# B&R Automation Studio project NAEUL004C00R13L518F00 (part 6)

### Hardware
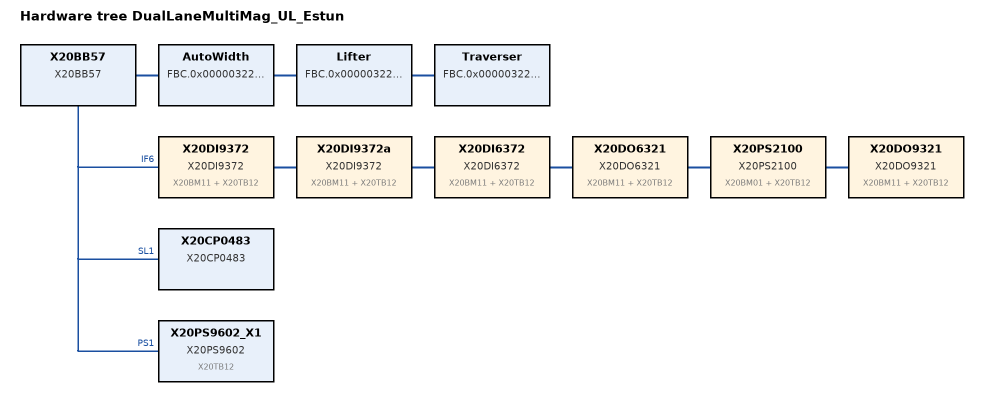
[picture p16: hardware tree DualLaneMultiMag_UL_Estun]
```
AutoWidth : FBC.0x00000322.0x00001000.NUTEK_ESTUN_PronetPlus_EDS_V106 v1.06.1 (OrderNumber=NUTEK_ESTUN_PronetPlus_V106)  [CAN1 -> X20BB57.IF7 (NodeNumber=16)]
Lifter : FBC.0x00000322.0x00001000.NUTEK_ESTUN_PronetPlus_EDS_V106 v1.06.1 (OrderNumber=NUTEK_ESTUN_PronetPlus_V106)  [CAN1 -> AutoWidth.CAN2 (NodeNumber=17)]
Traverser : FBC.0x00000322.0x00001000.NUTEK_ESTUN_PronetPlus_EDS_V106 v1.06.1 (OrderNumber=NUTEK_ESTUN_PronetPlus_V106)  [CAN1 -> Lifter.CAN2]
X20BB57 : X20BB57 v1.1.1.0
  Connector IF1:
    Baudrate = 9600
    Parity = N
  Connector IF7:
    Baudrate = 1000000
    ActivateCanOpen = 1
    p100c_parametervalue = 1000
    p100d_parametervalue = 3
X20BM01 : X20BM01 v2.1.0.0  [X2X1 -> X20BM11e.X2X2]
X20BM11 : X20BM11 v1.0.0.1  [X2X1 -> X20BB57.IF6]
X20BM11a : X20BM11 v1.0.0.1  [X2X1 -> X20BM11.X2X2]
X20BM11b : X20BM11 v1.0.0.1  [X2X1 -> X20BM11a.X2X2]
X20BM11e : X20BM11 v1.0.0.1  [X2X1 -> X20BM11b.X2X2]
X20BM11f : X20BM11 v1.0.0.1  [X2X1 -> X20BM01.X2X2]
X20CP0483 : X20CP0483 v1.2.1.0  [SL -> X20BB57.SL1]
  Connector IF2:
    ActivateDevice = 1
    Mode = Manual
    InternetAddress = 192.168.0.14
    SubnetMask = 255.255.255.0
    InaNodeNumber = 14
    Vnc1
    VncVcObjectName1 = Visu
    VncKeyMappingFile1 = 
    VncMaxConnections1 = 3
    VncRefreshRate1 = 100
    ActivateSnmp = 2
  ConfigurationID = NAEUL004
  VolatileGlobalPvSize = 80000
  EnableUsbRemoteInstall = 1
  TimerDeviceType = SWIOTIMER
  Cyclic1Duration = 10000
  Cyclic1Tolerance = 10000
  Cyclic2Duration = 20000
  Cyclic2Tolerance = 20000
  Cyclic3Duration = 50000
  Cyclic3Tolerance = 50000
  Cyclic4Duration = 10000
  Cyclic4Tolerance = 10000
  Cyclic5Duration = 200000
  Cyclic5Tolerance = 200000
  Cyclic6Duration = 500000
  Cyclic6Tolerance = 500000
  Cyclic7Duration = 1000000
  Cyclic7Tolerance = 1000000
  Cyclic8Duration = 10000
  Cyclic8Tolerance = 10000
  FileDevice1
  FileDeviceName1 = C
  FileDevicePath1 = C:
  FileDevice2
  FileDeviceName2 = User
  FileDevicePath2 = C:\User
  FileDevice3
  FileDeviceName3 = Private
  FileDevicePath3 = C:\Private
  FileDevice4
  FileDeviceName4 = CustomerUser
  FileDevicePath4 = C:\User\UserMgmt
  FileDevice5
  FileDeviceName5 = ProdRcp
  FileDevicePath5 = C:\User\ProductRecipe
  FileDevice6
  FileDeviceName6 = MagRcp
  FileDevicePath6 = C:\User\MagazineRecipe
  FileDevice7
  FileDeviceName7 = Alarm
  FileDevicePath7 = C:\User\Alarm
  FileDevice8
  FileDeviceName8 = McParam
  FileDevicePath8 = C:\User\MachineParameter
  FileDevice9
  FileDeviceName9 = NtParam
  FileDevicePath9 = C:\Private\NutekParameter
  FileDevice10
  FileDeviceName10 = LibVer
  FileDevicePath10 = C:\User\LibrariesVersion
  FileDevice11
  FileDeviceName11 = Retain
  FileDevicePath11 = C:\User\Retain
  FileDevice12
  FileDeviceName12 = Log
  FileDevicePath12 = C:\User\Log
  FileDevice13
  FileDeviceName13 = LCS
  FileDevicePath13 = C:\User\LCS
  FileDevice14
  FileDeviceName14 = MpProdRcp
  FileDevicePath14 = C:\User\ProductRecipeXml
  FileDevice15
  FileDeviceName15 = MpNtParam
  FileDevicePath15 = C:\Private\NutekParameterXml
  FtpUser1
  FtpUsername1 = NTAFTP
  FtpUserPassword1 = +UZ5u8Axw7KkkY4oM/r7wOOfB5oWHxpSY6r3j++jJso=  // NTA4BH
  FtpUserSalt1 = c0Alfi1W
  FTPAccessRight1 = 0
  FTPdevice1 = ALL
  FtpUser2
  FtpUsername2 = admin
  FtpUserPassword2 = mW+qRsE1LOSFDAB60rBJwb9dZ7uQUIuoHZp04C+x5XU=  // admin
  FtpUserSalt2 = Nr9+IHjr
  FTPAccessRight2 = 0
  FTPMSPartition2 = SYSTEM
  FTPMSpath2 = User
  FtpUser3
  FtpUsername3 = LCS
  FtpUserPassword3 = W4lkF6NjcyaB1sRdLwIoSAlqHoAE4GimWQdq7pKTzbA=  // LCS
  FtpUserSalt3 = f3H7b7h0
  FTPMSPartition3 = SYSTEM
  FTPMSpath3 = User\LCS
  ActivateOpcUa = 1
  OpcUa_ConversationSecurityPolicy_EnableBasic256Rsa256 = 0
  OpcUaInformationModels_PV_Version = 1
X20DI6372 : X20DI6372 v1.1.0.0  [SS1 -> X20TB12c.SS; SL -> X20BM11b.SL1]
X20DI9372 : X20DI9372 v1.1.0.0  [SS1 -> X20TB12a.SS; SL -> X20BM11.SL1]
X20DI9372a : X20DI9372 v1.1.0.0  [SS1 -> X20TB12b.SS; SL -> X20BM11a.SL1]
X20DO6321 : X20DO6321 v1.1.0.0  [SS1 -> X20TB12f.SS; SL -> X20BM11e.SL1]
X20DO9321 : X20DO9321 v1.1.0.0  [SS1 -> X20TB12h.SS; SL -> X20BM11f.SL1]
X20PS2100 : X20PS2100 v1.2.0.0  [SS1 -> X20TB12g.SS; SL -> X20BM01.SL1]
X20PS9602_X1 : X20PS9602 v1.0.2.0  [PS -> X20BB57.PS1; SS1 -> X20TB12.SS]
X20TB12 : X20TB12 v1.0.0.0
X20TB12a : X20TB12 v1.0.0.0
X20TB12b : X20TB12 v1.0.0.0
X20TB12c : X20TB12 v1.0.0.0
X20TB12f : X20TB12 v1.0.0.0
X20TB12g : X20TB12 v1.0.0.0
X20TB12h : X20TB12 v1.0.0.0
```

## Logical view

Binary libraries used (declarations not repeated): standard, runtime, astime, asstring, operator, AsIecCon, AsCANopen, visapi, FileIO, AsIODiag, AsMem, dvframe, AsOpcUac, AsARCfg, sys_lib, AsTCP, AsFltGen, brsystem, MpCom, MpBase, MpRecipe, Acp10man, Acp10par, NcGlobal, AsMath, NtBuffer, NtConv, NtFileIO, NtLogFile, NtMem, NtMessage, NtOvenInfo, NtPneu, NtRS232, NtSMEMA, NtTCP, NtTLBuz, NtVersion, NtSOT 5.00.0, NtLF, NtMotion, NtRecipe 5.00.5, NtHermes 5.00.4, NtOPCUA 5.00.1

### Update LogLibrary.txt
```
2023-09-06
NtOPCUA 6.01.0 - Add fbOPCUAMethodGetHandle and fbOPCUAMethodCall, updated fbOPCUAGetNodeHdlList

2023-05-22
NtHermes 5.00.4 Upgrade the Supervisory Hermes

2022-07-05
NtRecipe 5.00.4 Debug of Sorting Function

2022-01-25
NtRecipe 5.00.4 - Improve fRecipeNmCompare

2021-12-29
NtLF 5.01.5 - Add bDBAOnWOAlign to send DBA even width check sensor is not aligned.

2021-10-19
NtMotion 5.00.9 - Uncheck servo on and homing operation if both have been done.

2021-09-30
NtHermes 5.00.4 - Hermes v1.3

2021-09-01
NtLF 5.01.4 - Modify Product Recipe Name Related Variables to STRING[254].
NtUSB 5.00.5 - Add bEn := false for each fb when they are idling.

2021-07-08
NtUSB 5.00.4 - Improve fbDecodeStdKey.Changed ReadIdx Size, Check Array Limit.

2021-06-28
NtUI 5.00.2 - Add tyUIBitmap & tyUIBtn (uiValueIdx) to accomodate higher range of bitmap offset index

2021-04-20
NtLF 5.01.3 - Update fLFUSAllow & fLFDSAllow Block Conditions
			- Modify fLFFollowerProdAccDataReq.

2021-02-26
NtSMEMA:5.00.6 - Add fbSMEMATransporting1 for DS
NtLF:5.01.2 - Two Modes For Sequential. Modify fLFUSAllow For 3rd Party Usage.

2021-02-24
NtLF:5.01.2 - Modify fLFUSAllow.

2021-02-17
NtMotion 5.00.8 - Limit sensor interlock for Estun Servo Movement. (20210217)
       - Homing timeout in 3 sec if home sensor broken.
       - Set default value for servo parameter if the NtParam setting out of the limit.

2021-02-24
NtLF:5.01.2 - Modify fLFUSAllow.

2021-02-21
NtSMEMA: 5.00.6 - Add fbSMEMATransporting1.

2021-02-17
5.00.8 - Limit sensor intelock for Estun Servo Movement. (20210217)
       - Homing timeout in 3 sec if home sensor broken.
       - Set default value for servo parameter if the NtParam setting out of the limit.

2021-02-05
NtSMEMA:5.00.5 - Update fbSMEMATransporting

2020-11-14
NtUSB 5.00.0 - New Library Design.

2020-11-10
NtMotion:5.00.7 - Torque limit setting at NtParam.

2020-10-05
NtLF:5.01.1 - Improve Change All For Section Leader, Debug Change Sequential.

2020-09-10
NtTCP:5.00.2 - Change of fbTCPClntConnect.

2020-08-17
NtVersion:5.01.1 - Change of fChkFileValidity & fInvalidCharInFileChk to function block.

2020-08-06
NtLF:5.01.0 - Improve leader follower concept.
			- Add more tags in tyLeaderToFollowerTag and tyFollowerToLeaderTag.
NtVersion:5.01.0 - Add fChkFileValidity and fInvalidCharInFileChk.

2020-07-24
NtRecipe:5.00.3 - Debug of sorting functions.

2020-06-30
NtMotion:5.00.6 - Homing action when remote side limit sensor is on.

2020-06-15
NtMotion:5.00.5 - Homing timeout error when limit switch disconnecte.

2020-06-08
NtRecipe:5.00.2 - Update Product Recipe to 254, Add Sorting and End Character Filter Functions.
NtVersion:5.00.1 - Debug of fChkLibrariesVer.

2020-06-07
NtUI:5.00.1 - Update fbTableCtrl and fbTableCtrl_v2. Update tyUILString.

2020-06-01
NtStepper:5.00.0  - New Release.
NtConv:5.00.3	  - Added fbConvSenToSenBrkTm2Lmt & fbConvSenToSenBrk2.

2020-03-20
NtMotion - Add Estun Pronet, Schneider Electric Lexium 28 Servo Motor Control.
		- Resolve Limit Switch Alarm when Delta servo motor perform homing at stratup of auto mode.
NtParam - Add the selection of Motor model.

2020-03-16
NtTLBuz - Add inputs to allow repeat sequence for fbTLBuzWarn.
TLBuz - Add two inputs for buzzer behaviour, towerlight flash function to act_background and reset fbwarning.

2019-12-24
NtLF - Modify fbLeaderBlkDS, include machine index before & after oven 2, block machine to machine when different width
LFLeader - Remove fbBlkDS2 in Act_Initial & Act_Background_Process, add pa_bLFOnline in Act_Background_Process

2019-10-31
TLBuz - Regroup Structure Into Nutek, Aptiv & MEK.
MagConv - Separate Program Into MagConv1Clamper & MagConv2Clamper.

2019-10-29
NtHermes - Debug of fHermesGetTimeStamp

2019-10-21
NtRecipe - Debug Of fRecipeGetInfo.
NtSMEMA - fbSMEMAUS_9851, fbSMEMAUS_Std, fbSMEMADS_OppFirst, reset signal while error.
NtBuffer - Debug of fBffrSetFull, fBffrSetMty for slot disable.
NtLF - Add bBypassMnlAccDat Tag Name, Improve Change All Function Without Manually Accept Data.
MagConv - Improve with Action MagConvActPreExit & MagConvActPreExitClpr.
LFFollower - Improve Change All Function Without Manually Accept Data.
LFLeader - Add Second Oven Index, Improve Change All Function Without Manually Accept Data.
OpcUaMap.uad - Enable bBypassMnlAccDat Tag Name.
Startup - Act_Main_SDOWrite, Remove SDOWrite.
CANOpenServo - Change Structure Of SDOWrite And Abnormal Movement.

2019-07-30
NtMotion - Add Input To Select Homing Without Index Pulse.
CANOpenServo - Due To Upgrade of NtMotion.

2019-07-19
NtSMEMA - fbSMEMADS, reset signal while error.

2019-07-18
LFFollower - Act_Link, Minor debug.

2019-07-15
LCS - Act_Link, Check Recipe Name Must Not Exceed 15 Char.

2019-07-10
LCS - Add More Parameter For Live Data.

2019-07-04
LFFollower - Improve of Recipe Compare Method For p_tyInternalReqProdRcp, tyUpdtProdRcp & tyRlsBrdProdRcpNm.

2019-07-03
LFFollower - Improve Act_Background To Check Whole Product Recipe Different Instead of Name & Width Only.
Buffer - Add p_tyBufferStat & p_tyDispBuffer And Improve For Two Program Control One Memory.
NtBuffer - Debug Of Limit Buffer Range.

2019-06-28
USHermes - Improve of Act_Background_AccData.
DSHermes - Move of Act_Background_ChgConfig.
Buffer - Improve of bParamDiff Condition.
LCSLF - Improve of LCSActRunProd.

2019-06-27
LFFollower - Improvement To Change Name & Width To Whole Product Recipe Type.

2019-06-17
Conv - Add Two Action : ConvActEntToInOff & ConvActRevImmedStart.

2019-06-12
LFFollower - Add Act_Background_ChkRlsBrd. Improvement of Act_Background_UpdtData.
LCSLF - Add Update Data in Act_Background.

2019-06-11
TLBuz - Modify ChgRcp.
LFFollower - Improvement of UpdtData.

2019-06-10
ProdRcp - Update tyCurrRcp To a_tyCurrRcp (Array).
LFFollower - Add p_bInternalUse.
USHermes - Add p_bInternalUse.
DSHermes - Add p_bInternalUse.

2019-06-07
NtTLBuz - Improve of fbTLBuzWarn.
TLBuz - Add Warning & ChgRcp.
TCP - Add Start Code & End Code Checking.
Buffer - Improve bParamDiff. Add bFIFOOld.

2019-06-04
USHermes - Improvement At Accept Date (Act_Background_AccData).

2019-06-02
TCP - New.

2019-05-30
Hermes - Debug CheckAlive. SequenceTO Start Only After Connection Establish.
NtSMEMA - Improve fbSMEMATransportIdle.
Flatstream - Debug Act_Main.
USHermes - Update Act_Link to Accept New Recipe.

2019-05-29
NtRS232 - Add Flatstream Function.
DVFrame - Change From RS232. Improvement & Debug.
Flatstream - New.

2019-05-28
MagConv - Add MagConvActInitClpStop.
DCConv - Improvement of DC Motor Alarm Trigger Time.
LFFollower - Improve of Act_Background.
NtBuffer - Debug of fBffrNxtLoadNearby.
LCS - Add "Warning" & "Info" For Live Data.

2019-05-27
LFFollower - Debug Act_Link.
LCS - Debug Act_Link. Add sErrMsg.
Buffer - Debug Act_Main_Bffr. Add bMagRemoved.
Data - Update of Default User.dat.

2019-05-24
LFFollower - Improve of Act_Background.
MagConv - Add MagConvActEntClpStop.
TLBuz - Modify Warning Condition.

2019-05-22
NtLF - ChgAll Will Bypass Width Check Sensor.
OpcUaMap.uad - Update Tag Name.
LF - Modify Set Time. Improve Of Act_Background for Accept Data.
LFLeader - Add New Tag Name.
Time - Update of Act_InitGlobal For LF Sync Time.
LCS - Update To Reset If Receive Idle From LCS.

2019-05-21
NtRS232 - Add fbFullReadUntilValid.
RS232 - Add FullReadUntilValid.
LCS - Move Some Program From Act_Background To Act_Link. Bug Fixed.

2019-05-20
RS232 - Modify to work with start code & end code.
ProdRcp - Modify on dtLastModified in Act_LinkAction.
LCS - Act_Background Show Boolean & dtLastModified Working Sample. Add Function Enable.
TLBuz - Add Aptiv Mode.
NtParam - Add eTLBuzMod.

2019-05-18
Buffer - Check Next Unload Ignore Product Name.

2019-05-17
NtMessage - Debug When Attribute Value Is Empty String.

2019-05-15
OvenInfo - Improve of Act_Background.
Buffer - Add bParamDiff to check current parameter and request parameter different.

2019-05-14
LCS - Update Act_InitGlobal.
RS232 - New.

2019-05-11
LFFollower - Improve And Able To Ignore MagRcp If Necessary.

2019-05-10
TLBuz - Add Simulation Mode.
ProdRcp - Improve Act_LinkAction.
Buffer - Improve Act_LinkAction.
HWInfo - Improve Act_Main While In Simulation.

2019-05-09
CANOpenServo - Improve of Error Axis Move Abnormally By External Force (10000).
ProdRcp - Debug Write Recipe. Add Save List.
MagRcp - Debug Write Recipe. Add Save List.
UsrFolder - Create LCS Directory.
Startup - Act_Main_UsrFolder, Create LCS Directory.
Alarm - Combine Two Alarm Info.

2019-05-08
RmtHermes - Debug Log title.
UsrMgmt - Add Access Right Output.

2019-05-07
NtConv - After Time Out, Reset Output.
MagConv - Debug.
ConvBffr - Add Individual Have Board Output.
NtLF - Debug fLFUSAllow. Modify fbLFFollower.
LF - Major update.
LCSLF - Change Name to tyCurrProdRcp.
ProdRcp - Add Write Recipe Parameter.
MagRcp - Add Write Recipe Parameter.
LCS - Update to match LCS (PC).

2019-05-04
MagRcp - Split Current Magazine Recipe From McParam.
ProdRcp - Split Current Product Recipe From McParam.
UsrMgmt - Split Access Right From McParam. Remove Nutek User.
Hermes - Split Configuration From McParam. Add RmtHermes.
Startup - Split Parameters From McParam. Add RmtHermes.
Remove "File Device" "NutekUser". Please Refer Configuration "4PPC30_043F_21F001".
NtHermes - Debug Due to RmtHermes.

2019-05-01
Hermes - Log file change to day instead of hour. Due to startup too long to check old log when production run for long.

2019-04-30
LCS - Improve To Match LCS (PC).
LFLeader - Make a_tyFollowerToLeaderTag as Output.
All - sStatTxt & a_sStatText Change To String[200].
ProdRcp - Modify For LCS.

2019-04-28
MpProdRcp - New.
Add "Config.mprecipexml" Under Configuration View > mapp. Please Refer Configuration "4PPC30_043F_21F001".
Add "File devices" For "MpProdRcp". Please Refer Configuration "4PPC30_043F_21F001".
Startup - Modify Due To MpProdRcp.

2019-04-27
NtSMEMA - Improve Standard SMEMA According to Nutek Standard.
DSSMEMA - Update due to NtSMEMA upgrade.

2019-04-26
Buffer - Debug tyBuffer to p_tyBuffer. Improve bLastProductUnload Condition In Unload Board.
Startup - Get Retain ConvBffr.
ConvBffr - Update Link with Startup. Improve bLastProduct Condition In Remove Board. Add Have Board Output.
LFFollower - Improve Act_LinkEn. Add Condition in Act_Link to update current recipe into leader tag.

2019-04-25
NtHermes - Debug fHermesIllegalMsgBrdAvlDS. To Handle MachineReady & StartTransport Send In One Message.
LibVer - Modify To Move LibVer From "Private" To "User".
Update "File devices" For "LibVer". Please Refer Configuration "4PPC30_043F_21F001".
Add "File devices" For "LCS". Please Refer Configuration "4PPC30_043F_21F001".
Modify "FTP Server" "Users". Please Refer Configuration "4PPC30_043F_21F001".
Modify "OpcUaMap.uad". Please Refer Configuration "4PPC30_043F_21F001".
LFLeader - Improvement.

2019-04-24
CANOpenServo - Add actual limit sensor output.
ProdRcp - Add "Add" & "Edit" action. Improve of Act_LinkAction to suit LCS.
LCS - New.

2019-04-23
NtLF - Major upgrade.
LFLeader - New.

2019-04-21
USHermes - Modify Alarm Info.
LFFollower - New.

2019-04-18
ConvBffr - New.
NtBffr - Add Buffer Name, Product Name & Barcode.
Buffer - Change of NtBffr.

2019-04-17
CANOpenServo - Remove Extra Homing Parameter, All Use Under tyMotionCANParamInHm.

2019-04-16
Operations - Remove Accept Data & New Data.
Hermes - Debug Log File. Modify Accept Data.

2019-04-11
USHermes - Debug Log by adding step. Add p_bAccDataRdy.
DSHermes - Debug Log by adding step.
NtConv - Debug of Time Out Error.

2019-04-10
Startup - bNtSettingsLoadDone should be FALSE as default.

2019-04-09
Ops2 - Update of p_bAccDat interlock by Ops1.
USHermes - Update AccDatStep in Act_Link. Remove p_bChkBrdAvl. eStatus2 = Error then bRdyRcv = false. Update Act_Background_BoardAvailableChk. Add Manual Accept Data.
DSHermes - Make local.var BoardAvailable new board parameter to default value.
NtParam - Change of Act_LinkAction.
TLBuz - Change of Act_LinkAction.
Buffer - Change of Act_LinkAction.
Conv - Change of Act_LinkAction.
DCConv - Change of Act_LinkAction.
MagConv - Change of Act_LinkAction.
MotorBrk - Change of Act_LinkAction.
ConvSpd - Change of Act_LinkAction.
SMEMA - Change of Act_LinkAction.
Pneu - Change of Act_LinkAction.
CANOpenServo - Change of Act_LinkAction.
Hermes - Change of Act_LinkAction.

2019-04-08
DSHermes - Minor debug on fbParseBrdAvlExternal.
Hermes - Add program Hermes for board available memory use.
Startup - Due to change of Hermes.

2019-04-04
OvenInfo - Add p_bBGRun.
NtBuffer - Modify fBffrStat.
Startup - Change eStartupStep member order for better display in UI.
UsrMgmt - Add UsrMgmtActUsrBypassLogin & UsrMgmtActNtBypassLogin.
DSHermes - Debug BoardAvailable for "New" and "External".
UI - Remove Not Use Page.

2019-04-02
NtTCP - fbTPCSend & fbTCPRcv modify bEn = False condition. Disable check alive set function in Simulation Mode.

2019-03-29
All - Add Act_LinkAction.

2019-03-28
Startup - Change "DelOldLogFile" to "Alarm". Add "Hermes". Error will reset Action to IDLE.

2019-03-25
All - Change Action become input. Merge Alarm Text & Recovery Text into one type.
NtGeneral - Add tyAlmTxt.
NtLogFile - Increase Alarm String Size.

2019-03-22
Startup - Add bNtSettingsLoadDone. Move StartupStepParameter after StartupStepUsrFolder in Act_Main.st.
All - Update to match latest method of NtParam.

2019-03-16
Startup - Act_Main_Bffr. Add BufferActBGStartCoolFan in Step 8.

2019-03-15
NtHermes - New Release
Hermes - New Release

2019-03-13
UsrFolder - Debug of Log directory path. Add "FileDevice" for "Log".

2019-03-11
DCConv - Minor debug.

2019-02-26
AWClose - Minor debug.

2019-02-23
Alarm - Minor debug.
UsrFolder - Add Create Log Directory.
Startup - Improve of "Act_Main_UsrFolder" due to UsrFolder update.

2019-02-22
CANOpenServo - Change of Act_Action.

2019-02-21
DOutput - Add Act_Link.

2019-02-20
DCConv - Debug of ConvEngage.
NtMotion - Update to 5.00.1. Update LibrariesVersion.dat.
CANOpenServo - fbModuleOK delay time change to 5s.

2019-02-19
CANOpenServo - Reset Error need to reset control word 6040.
TLBuz - Improve of condition while p_bManual = True.

2019-02-18
Buffer - Add background control of cool fan run.

2019-02-15
Conv - Improve of condition while p_bManual = True.
DCConv - Improve of condition while p_bManual = True.
MagConv - Improve of condition while p_bManual = True.
MotorBrk - Improve of condition while p_bManual = True.
SMEMA - Improve of condition while p_bManual = True.

2019-02-14
ConvSpd - Improve of condition while p_bManual = TRUE.
Change of Cyclic Time.
NtMotion - Change of Position Different Threshold.
CANOpenServo - Change of Position Different Threshold.
Convert Library Into Binary

2019-02-11
TLBuz - Warning Rest Time Change To 5s.
Buffer - Add Magazine Present Timer.

2019-01-27
Buffer - Add error code.

2019-01-26
Buffer - Debug.

2019-01-25
Buffer - Debug a_bSkip array size.
Lifter - Debug Act_Background.
User.dat & NtUser.dat update.

2019-01-24
Pneu - Modify Cyclic for disable.
AW - Add GoWidthOff to turn off motor after auto width move.
Lifter - Debug.
Traverser - Debug.
Buffer - Debug. Add background update display.
OvenInfo - Modify Act_Main_Disable.

2019-01-23
Lifter - Major debug in slot calculation. Add FullMovRel.
CANOpenServo - Debug reset error. Debug Act_Alarm.
DCConv - Debug reset error.
Machine - Debug reset error.
Operation - Debug reset error.

2019-01-22
CANOpenServo - Minor debug.

2019-01-21
DInput - Debug reset error.
CANOpenServo - Add eMainStatus. Add bJogging.
NtMotion - Update fbMotionModuleOK.
Time - Add eMainStatus.
Operations - Rename eStatus & udiStatus.

2019-01-20
Operations - Update Structure.
NtSMEMA - Update.
SMEMA - Update due to Library update.
Buffer - Add error code.

2019-01-19
TLBuz - Add Warning.

2019-01-18
RstErr - Act_Main update.
NtMotion - Update for FwdLimit & RevLimit.
CANOpenServo - Add output. Set Default Value for siModOfOptDisp_6061:=6.
Change of Cyclic time.
Buffer - Update Local.var
Add file for NtUser, LibrariesVersion & User.
Conv - Add Pneu status output.
DCConv - Add Pneu status output.
Operations - Modify structure in Cyclic.

2019-01-17
DCConv - Act_Main debug.

2019-01-16
Trav - Remove diPitch.
Lifter - Remove diPitch.
Operations - Modify Reset methos.

2019-01-15
McParam - File name as input.
NtParam - File name as input.
Buffer - File name as input.
Operations - Add bAccData.

2019-01-14
Operations - Update Alarm & Sequence.
SMEMA - bTimer & bVirtual as output. Debug Act_Background timer interlock.

2019-01-12
Conv - Convert time out type.
DCConv - Convert time out type.
MagConv - Convert time out type.
OvenInfo - diBrdInOven change to retain.
SMEMA - Update timer condition. Add bComplSigOn.
Startup - Debug for HWInfo.

2019-01-11
NtSMEMA - Update library.
SMEMA - Minor debug. Add Act_LinkEn.
Operations - Add alarm. Add Act_LinkEn.
MagRcp - Add Act_LinkEn.
OvenInfo - Add Act_LinkEn. Minor debug.
Conv - Add Act_LinkEn. Add conveyor time out.
DCConv - Add Act_LinkEn. Add conveyor time out.
MagConv - Add Act_LinkEn. Add conveyor time out.
MotorBrk - Add Act_LinkEn.
ConvSpd - Add Act_LinkEn.
RS232Mirtec - Add Act_LinkEn.
Pneu - Add Act_LinkEn.
CANOpenServo - Add Act_LinkEn. Major Update.
NtConv - Add time out.

2019-01-10
McParam - Remove ProdRcpWrite & MagRcpWrite.
OvenInfo - Act_Main modify for change of eStat.
Conv - Act_Main modify for change of eStat.
DCConv - Act_Main modify for change of eStat.
MagConv - Act_Main modify for change of eStat.
MotorBrk - Act_Main modify for change of eStat.
ConvSpd - Act_Main modify for change of eStat.
SMEMA - Act_Main modify for change of eStat.
DOutput - Act_Main modify for change of eStat.
Pneu - Act_Main modify for change of eStat.
Operations - Act_Main modify for change of eStat.

2019-01-09
AW - Update bWidthPosDiff when disable.
Lifter - Update bSltPosDiff when disable.
NtMotion - Debug move absolute with backlash.
Conv - Add bGdBrdInit. Debug tMtrOffDlyTm. Improve Act_Action to let eStatus = DONE also able change eStat directly.
DCConv - Add bGdBrdInit. Improve Act_Action to let eStatus = DONE also able change eStat directly.
SMEMA - Add tRstDlyTm. Improve Act_Action to let eStatus = DONE also able change eStat directly.
Operations - Add Act_Main_Disable. Improve Act_Action to let eStatus = DONE also able change eStat directly.
TLBuz - Improve Act_Action to let eStatus = DONE also able change eStat directly.
OvenInfo - Improve Act_Action to let eStatus = DONE also able change eStat directly.
MagConv - Improve Act_Action to let eStatus = DONE also able change eStat directly.
MotorBrk - Improve Act_Action to let eStatus = DONE also able change eStat directly.
ConvSpd - Improve Act_Action to let eStatus = DONE also able change eStat directly.
DOutput - Improve Act_Action to let eStatus = DONE also able change eStat directly.
Pneu - Improve Act_Action to let eStatus = DONE also able change eStat directly.

2019-01-08
NtMotion - Debug move absolute with backlash.
NtConv - Debug end sensor edgeneg trigger.
DOutput - Add output.
SMEMA - bTimer will be trigger only during SMEMAActRun.
Operations - Combine Ops1 & Ops2 into Ops.

2019-01-07
SMEMA - Add bUSRdy, bUSGdBrdRdy & bDSRdy for USSMEMA & DSSMEMA.
Conv - Add tMtrOffDlyTm.
DCConv - Add tMtrOffDlyTm.
MagConv - Add tMtrOffDlyTm.
Time - Combine Error
CANOpenServo - Combine Error
Alarm - Remove link data.

2019-01-04
Machine - Debug Act_Alarm1.
Time - Debug Init.st.
Operations - Debug Ops1 > Act_Main. Add sStepTxt into Act_Main. Add Act_Dummy.
NtConv - Add fbConvSenToSenOff1.
Conv - Due to NtConv update, add one more type of Exit.
DCConv - Due to NtConv update, add one more type of Exit.
MagConv - Due to NtConv update, add one more type of Exit.
SMEMA - Add Timer & Virtual.

2019-01-03
Machine - Debug Act_Alarm & Act_Alarm1. Modify background error handling.
CANOpenServo - Modify background error handling. Update sStatTxt in Act_Initial.
AW - Replace diStandPitchInUM (Input) to diPitchInUM (Local).
Time - Modify background error handling. Update sStatTxt in Act_Initial.
DCConv - Modify background error handling. Update sStatTxt in Act_Initial.
DInput - Modify background error handling.
UsrMgmt - Update sStatTxt in Act_Initial.
McParam - Update sStatTxt in Act_Initial.
NtParam - Update sStatTxt in Act_Initial.
ProdRcp - Update sStatTxt in Act_Initial.
MagRcp - Update sStatTxt in Act_Initial.
HWInfo - Update sStatTxt in Act_Initial.
UsrFolder - Update sStatTxt in Act_Initial.
LibVer - Update sStatTxt in Act_Initial.
General - Update sStatTxt in Act_Initial.
TLBuz - Update sStatTxt in Act_Initial.
OvenInfo - Update sStatTxt in Act_Initial.
Buffer - Update sStatTxt in Act_Initial.
RstErr - Update sStatTxt in Act_Initial.
Conv - Update sStatTxt in Act_Initial.
MagConv - Update sStatTxt in Act_Initial.
MotorBrk - Update sStatTxt in Act_Initial.
ConvSpd - Update sStatTxt in Act_Initial.
Alarm - Update sStatTxt in Act_Initial.
RS232Mirtec - Update sStatTxt in Act_Initial.
SMEMA - Update sStatTxt in Act_Initial.
UI - Update sStatTxt in Act_Initial.
DOutput - Update sStatTxt in Act_Initial.
Pneu - Update sStatTxt in Act_Initial.
Operations - Update sStatTxt in Act_Initial.
Startup - Update sStatTxt in Act_Initial.
NtTCP - Update.
NtMessage - Update.

2019-01-02
UsrMgmt - Change of sStatTxt update.
McParam - Change of sStatTxt update.
NtParam - Change of sStatTxt update.
ProdRcp - Change of sStatTxt update.
MagRcp - Change of sStatTxt update.
Time - Change of sStatTxt update.
HWInfo - Change of sStatTxt update.
UsrFolder - Change of sStatTxt update.
LibVer - Change of sStatTxt update.
General - Change of sStatTxt update.
TLBuz - Change of sStatTxt update.
OvenInfo - Change of sStatTxt update.
Buffer - Change of sStatTxt update.
RstErr - Change of sStatTxt update.
Conv - Change of sStatTxt update.
DCConv - Change of sStatTxt update.
MagConv - Change of sStatTxt update.
MotorBrk - Change of sStatTxt update.
ConvSpd - Change of sStatTxt update.
Alarm - Change of sStatTxt update.
RS232Mirtec - Change of sStatTxt update.
SMEMA - Change of sStatTxt update.
UI - Change of sStatTxt update.
DOutput - Change of sStatTxt update.
Pneu - Change of sStatTxt update.
Operations - Change of sStatTxt update.
CANOpenServo - Change of sStatTxt update. Update eStatus to Busy while running.
Startup - Change of sStatTxt update.

2018-12-31
CANOpenServo - Seperate input reference.

2018-12-27
Time - Remove bBGRun.
TLBuz - Remove bBGRun. Add manual reset.
OvenInfo - Background direct link to input bPrepExtdd, bEnExtdd & bDisExtdd. Add manual reset.
Buffer - Background Cool Fan Control direct link to input bPrepCoolTm & bCoolFanTm.
DCConv - Remove bBGRun. Add manual reset.
AlarmLog - Background run is control by Action.
Machine - Remove bBGRun.
SMEMA - Remove bBGRun. Add manual reset.
DInput - Remove bBGRun.
DOutput - Remove bBGRun. Add manual reset.
CANOpenServo - Remove bBGRun. Background run is control by Action. Add manual reset.
AW - Add bWidthPosDiff.
Lifter - Add bSltPosDiff.
Startup - Background run is control by Action. Shorten local variable name.
McParam - Add McParam program without Magazine (McParam2).
RstErr - Add manual reset.
Conv - Add manual reset.
MagConv - Add manual reset.
MotorBrk - Add manual reset.
ConvSpd - Add manual reset.
Pneu - Add manual reset.

2018-12-26
CPU - Update distribute of program in CPU. Update cyclic time.
FTP - Update of FTP server configurations.
Startup - Remove bStartupErr.
HWInfo - After set new IPAddr & Subnetmask will update output.
TLBuz - Rising of bManual will set Amber Light ON.
Conv - Remove functions reset in individual eStat.
MagConv - Remove functions reset in individual eStat.
MotorBrk - Remove functions reset in individual eStat.
DCConv - New program.
Operations - Update of OperationsActStep.

2018-12-24
Operations - Add bRun.Sequence will execute base on bRun instead of bStatusRun.

2018-12-21
Buffer - Add individual cooling fan control.
McParam - Move Hermes parameter to Hermes program type.
MagConv - Add bClprTwoOutputControl. Remove bClprUnclampCtrl.

2018-12-20
TLBuz - Add bMuteBuz.
OvenInfo - Add bDis.
Conv - Add bEn.
MagConv - Add bEn.
MotorBrk - Add bEn.
ConvSpd - Add bEn.
RS232Mirtec - Add bEn.
SMEMA - Add bDis.
Pneu - Add bEn.
CANOpenServo - Add bEn.
CANOpenServo - AutoWidth - Add diMaxWidthInUM, diMinWidthInUM, diWidthOffsetInUM & diStdPitch.
Operations - Add bPrep, bEn & bDis. Add OperationsStatusCycleStopping. Default Status is OperationsStatusStop. Add Boolean output for Status.
MagRcp - Change sDisplayInfo & Magazine Parameter.
Startup - Add bRun.

2018-12-14
RstErr - Add bManual to control reset of output in Idle. Reset output in Idle after ManualMode off.
Conv - Add bManual to control reset of output in Idle. Rename eAction. Reset output in Idle after ManualMode off.
ConvSpd - Add bManual to control reset of output in Idle. Reset output in Idle after ManualMode off.
MtrBrk - Add bManual to control reset of output in Idle. Rename eAction. Reset output in Idle after ManualMode off. Reset after change eStat.
MagConv - Add bManual to control reset of output in Idle. Rename eAction. Reset output in Idle after ManualMode off. Reset after change eStat.
OvenInfo - Set bOvenAllow to TRUE, if all functions not activated.
SMEMA - Reset output in Idle after ManualMode off.
Pneu - Add Extended & Retracted output.

2018-12-13
Conv - Change of Conv2Sen to Conv. Add Reject & Inspection functions. Add individual output control.
Pneu - Add bTwoCtrlIn & bTwoCtrlOut.
TLBuz - Add individual output control.
ConvSpd - Add individual output control.
OvenInfo - Add individual output control. Move functions into Act_Background.
RstErr - Add individual output control.
MtrBrk - Add individual output control.
MagConv - Add individual output control.
DOutput - Add individual output control.
SMEMA - Add individual output control.

2018-12-12
Startup - Add Logout during User Management Startup.
Time - Move Act_Background above Act_Main.
Buffer - Move Act_Background above Act_Main.
Alarm - Move Act_Background above Act_Main.
CANOpenServo - Move Act_Background above Act_Main.
Operations - Change of Conv2Sen to Conv.

2018-12-11
DOutput - Split to Act_InitGlobal & Act_InitLocal.
Pneu - Change in all program. Add Pneu3Sen program.
Operations - Update sample to 2 operations. Rename variable.
CANOpenServo - Rename variable.
```

### Update LogProgram.txt
```
5/1/2024 (R14)
-change configuration global memory to 50000
-lifter magazine platform can jog up while sensing safetylimitsensor

4/12/2023
 - mtr pusher use p_bTorqueSig to slow

23/11/2023
- Traverses need to react as soon as Lifter moving in Magazine Platform model
- Pneu2SenOutShutter , Act_LinkAction comment, lifter moving allow open or close shutter
- Lifter, iLifterMovedSlot
- TravLifULStepTravLifMov, p_bLocalDSRdy AND p_bDSAllow

21/11/2023
updated DefaultGate
Potential FileWrite IO
Added TravULStepClrSensorErrBefTrav, check clear and inlet sensor before traverse

2023-09-25, 11-1 (R13)
MagRcp - update reset MagRcp load single
CanOpen, Lifter and Traverser addd Interrupt sensor for inlet and clear sensor
DSSMEMA act-link , sendcompl make sure clr off
OpsTravLif - ExitBrd NOT(p_bConvClrSen OR p_bConvRgtSen)
			tExitBoardTimoutErr , Exit Brd Err when sensing
			- TravLifULStepExitBrd - added bSkipCloseInletShutter = false

2023-09-06
*CHANGE HMI IP ADDRESS Update*
McParam - Act_Link,Local.var, InputRef.var, Act_InitGlobal, Act_InitLocal, McParam.typ, Act_Initial, Act_Alarm
UI - Added Act_Background/P1021/Act_Opt1021HMIIpAddr, Local.var,Visu_Layer.typ, Visu_Page.typ, UI.var, Init, Act_Background/P1021/Act_Opt1021Save, Act_Background/Act_OptPage, Act_Main/Act_Main_p1021
Visu - AlarmGroups/Warning, TextGroups/T1010_TextRecovery, TextGroups/T1080_MachineSetting, P1021_MachineSettingGen/A1_General_1

2023-09-13
SMEMA p_bRdyRcv , p_bLinkOpsTravLifULUSComm
EntBrd at SMEMA stop , added p_eLocalUSSMEMAAct	:= SMEMAActIdle;
TravLifULStepStopperRet , TravLifULStepStopperExt include p_bLifterAPosDiff
MagConvULStepMagFullDSComm
p_bOutShutterExtended  changed to p_bDIOutShutterClosedRS3

2023-07-26
include Safety Relay Mute for after booting
Langauge Setting Layout adjust
LCS updated MagRcp Control (Havent prepared XML)
Deleting Lifter2 for smooth

2023-07-26
Debug for Manual Accept Data automatically accept after product change many times

2023-7-19
-Update Call for MES set magazine full (OPC UA)
-Release Magazine Will Wait the Board finished unloader
-Set Magazine Full immediately prevent the board entering(regardless of shutter open/close)
-Solved immediate Exit Magazine regardless shutter closing (SMEMA off)
-MagConvULStepBffrUSComm (bBffrFull)
-TravLifULStepTravLifMov(Shutter Retract only if p_bLocalDSRdy)
-ADDED bMagExitedWait to prevent fail magcmp

2023-07-13
-update Magazine BffrAvl Reset
-update Buzzer for AGV
-Update Oven Info, to Link to Rcp0 and MagPresent to cut off oven signal when no magazine present
-update when switch Horizontal Com Flush Magazine for Siemens
-update SMEMA not working

2023-06-23 (R12)
-Retain Memory on Traverser
-MagConv Error Handling (remove redudant Magazine Exit)

2023-6-22 (R11)
-Auto Rcp (Compatiple only with Horizontal Hermes 1.3)
- Magazine auto Calculated width,min,max,pitch based on Board Available and Board Forecast
- Magazine Properties Retain Function
-SvyHermes Board Arrived,Board depart (Slotid,Magazaine ID)
-OPCUA AGV with RFID, read RFID tag when enter, write when exit
-Adding Magazine Exiting with buffer full,release magazine, AGV ready signal , product different (Auto Rcp)
- Error Handling for AutoRcp

2023-5-18
Act_OpsRun.st (R10)
- TravLifULStepEntBrd,TravLifULStepInletPneuOpn,TravLifULStepTravLifMov,TravLifULStepUSSigRechkTwice
- added p_bLifterAPosDiff = FALSE
-when recover from DS to USSig to TravLifMov (Lane A close to Mag2), Lifter not moving
- added Alarm for AGV and MAG Conv
-TravULStepBrdLostInMiddle Error Prevent Potential Double feeding, Error occurred when Mid sensor miss out
-USSMEMAA & B Act_Link p_bComplSigOn changed to edge_neg (to alway check downpulse on inlet sensor)
-TravLifULStepEntBrd (McSetCommModSMEMA) changed to when finished SMEMA done close shutter then conveyor check done
-TravLifULStepEntBrd (McSetCommModHermes) [p_bLocalUSHermesStopTransport = TRUE, go close shutter]

2023 - 2 -15
Alarm
-Alarm.var added global variable to link text snippet alarm UI
-Act_Background - Recovery list changed to Alarm Error Code
-UI P0200 - change recovery text from string to text group
-UI P0600 - Trigger alarm using bAlm,bWarning,Errcode replacing the original string
-UI P0600 - Adding additional button to check alarm history
-UI Visu  - P0200,P0600 Using given Visu Alarm component instead of string text as the Alarm table

2022-11-3
- OpsTravLifUL    TravLifULStepInitAWTravLif ( p_bInShutDis = FALSE) changed to True to prevent shutter Open after initialized
- create Ntparm (eMidSenParam) in Dinput for ConMid to cater NC/NO type

2022-3-3
ProdRcp- Act_Main,Act_EntP1040Disp, Act_OptP1040Save,Act_OptP1040Del,Act_OptP1040ToXml,Act_OptP1040FromXml
MagRcp- Act_Main,Act_EntP1030Disp,Act_OptP1030Save,Act_OptP1030Del,Act_EntP0410Disp

2022-12-02 (R8)
-Add NtOpConXml (trace ability)
-Add Scanner feature ,top and bottom scannner
-UI optimization P0900
-magwidthchk for TopToBtm changed to slot 1 checking
-NtParam - Added tyPPTorqParam

2022-10-14 (R7)
- Add OutletShutter2Prep and OutletShutter3Prep for Lifter Magazine Platform
- TroubleShoot in OpsLifMagUL Script and OpsTravLifUL Script

2022-10-14 (R6)
- Added Pusher/Puller (servo)
- Added Curtain Sensor Feature
- Separated three Outlet shutter Control and RS
- Added Fix Clamp Magazine Detect sensor and two control

2022-05-24 (R4)
-Added dual lane magazine conveyor feature.

2022-05-11 (R3)
- LCS - Local.var - Add tyTagNm.sMcAlmMsg
-Background.st - Add Machine Alarm message to the opcUA.

2022-03-21 (R2)
LifterBtm - Act_Link - Set p_diMoveVelInUMPS to 50000 when magazine platform is used.

2022-02-23 (NAEUL004R1, L515)
UI - include dualmag (MagPlatform) outlet shutter image.
Configuration View - updated 23Mag_UL_LifterMagazinePlatform can be use in dual/ triple mag with same hardware module card.

2022-01-25 (NAEUL004R1, L515)
ProdRcp - Act_Main, Local.var
MagRcp - Act_Main, Local.var

2021-12-29
LFFollower, Follower1 - Act_Background - Add p_bDBAOnWOAlign to fbFolllower to send DBA even width check sensor is not aligned.

2021-10-19
CANOpenServo - Act_Background - Add error code for Estun Servo Motor.
			 - Reset control word 6040.4 to 0 when servo motor is in operation.

2021-12-01
Combine NAEUL100 and NAEUL003 software version into a software program.

2021-09-30
Hermes Program - Update
USHermes Program - Update
DSHermes Program - Update
RmtHermes Program - Update
SvyHermes Program - *NEW*
NtParam  - Add new variables for Hermes v1.3
McParam  - Update
Alarm - Update
Startup - Update
UI HMI & Program P0201 - Update
UI HMI & Program P1021 - Update
UI HMI & Program P1022 - Update
UI HMI & Program P1023 - Update

2021-09-02
Revision - R15 , L512
- Width Offset move to NtParam
- Add BadBrdRedLight in NtParam and P0200 for 2021-0532G.
- McMode2 for 2021-0532G in P0201,P0400,P1021,P1040
LFLeader, LFFollower - Local,Input_Ref variables - Modify Product Recipe Related Variables to STRING[254]
LFFollower - Act_Background - Modify bUSAllow To Include p_bInternalReqProdRcpDiff

2021-08-31
Revision - R14 , L512
LFFollower - Update Act_Background
Follower1 - Update Act_Background
- Update NtUSB to 5.00.5
- Update NtLF to 5.01.4
- OPC-UA Security Policy Basic256 Sha256 prohibited

2021-07-21
- Modbus Configuration
- Add usiMcBitmapIdx in NtParam
- Debug Act_Main_P1081 ManualFB, Act_OptP0935RstMnl & Act_OptP0936RstMnl.

2021-07-05
Revision - R13 , L510
- Update NtUI to 5.00.2

2021-06-28
Revision - R12
- Debug OpsInitGConv Act_Link
- Debug keypad title of Machine Index Before and After Oven

2021-06-14
Revision - R11
Add Good Bad Board and Taifun Sequence

2021-06-09
Revision - R10
Modify Act_Main_C0005 & Act_OptC0005ChgPage

2021-05-18
LFFollower - Act_Link - Change Info Message
		   - Act_Background, Act_Background_AccData - Change Product NameNot Exist and Width Mismatch Error To Info
		   - Act Main_Disable - Reset Variables When Function Is Disabled
Follower1  - Act_Background, Act_Background_AccData - Change Product NameNot Exist and Width Mismatch Error To Info
		   - Act Main_Disable - Reset Variables When Function Is Disabled

2021-04-20
Revision - R9
Alarm - Act_Background - Add bInfoLF.
LFLeader - Act_Main - remove input for sequential mode (one time or always active)

2021-02-18
Update - Visu - C0005
Update - UI - UI Folder - Act_Background - Act_OptC0005ChgPage.

2021-02-17
CANOpenServo - Act_Background - PosDiff updated from 50 to 500.
      			              - Remove condition udiStatus <> 10028.
	     - Act_Alarm - udiCode change to 10299
	     - Local.var - update alarm message a_tyAlmText[10298] and a_tyAlmText[10299]
	     - Act_Main - softwre update.
Teaching page add interupt sensor interlock for lifter and traverser.
Teaching page add Open and Close shutter button.
Magazine info screen display issue update.

2020-12-30
Clear sensor add into operation sequence.
Pusher retract after board stuck at outlet shutter side.

2020-11-11
Tuning.diAsdaA2FirstTorqueCmd default setting is 300 in NtParam for all Delta servo motor.
2020-10-05
Startup - Act_Main_GetHWInfo - Debug Steps In Network Recovering
LFLeader - Act_Initial, Act_Background_Process and Local.var - Rename and change the type of fbBlkUS to fbBlkUSDS
LFFollower, Follower1 - Act_Background, Act_Background_AccData - Add bLeaderOnline replacing the direct usage of tyLeaderInfo.bOnline
TLBuz - Add Buzzer For All Act_Backgrounds Change Manual Mode Towerlight To Cater For Error Indication
HWInfo - Act_Main - Add IF-ELSE Statement For Simulation, Update Alarm Code for fbGetETHConfigMode & fbSetETHConfigMode
		 Local.var - Add New Alarm Code fbGetETHConfigMode & fbSetETHConfigMode

2020-09-22
LFFollower - Reset bLeaderSeqCtrlInActive in Act_Main_Disable.
HWInfo.typ - Add One Enumeration (eNetworkConfigMod) & Two Actions (fbGetETHConfigMode and fbSetETHConfigMode) - Retrieve Or Set Network Configuration Of The PLC.
HWInfo Init, InitGlobal, InitLocal, Act Main, Act_Initial, Local.var and InputRef.var - Add The Additional Actions Related Variables
McParam  - McParam.typ Add eNetworkMod in tyMcParam.
NtParam  - NtParam.typ Add tyNetworkMOde (UILmt) in tyNtParam.
Startup	   - InitGlobal, InitLocal, Act_Main_GetHWInfo - Add Function To Load Saved Network Configuration s When New Configuration Detected.
		   InputRef_Link.var, InputRef.var & Local.var - Add New Startup Function Variables.

2020-09-16
McParam  - McParam.typ Add sIPAddr & sSubnetMask in tyMcParam.
Startup	 - Init, InitGlobal, InitLocal, Act_Main_GetHWInfo - Add Function To Load Saved IP Parameters When New IP Detected.
		   InputRef_Link.var, InputRef.var & Local.var - Add New HWInfo Function Variables.

2020-09-10
USHermes - Init, Cyclic, Act_Background_TCPConnect, Act_Alarm5 - Improvise Alarm For Connection Lost.
		   Local.var - Add New Alarm Variables & Modify Alarm Text.
DSHermes - Init, Cyclic, Act_Background_TCPListen, Act_Alarm4 - Improvise Alarm For Connection Lost.
		   Local.var - Add New Alarm Variables & Modify Alarm Text.

2020-08-17
LibVer - Act_Main - Modify Function To Function Block In LibVerActReadChk.
		 Act_Initial - Initialize Newly Added Function Blocks.
		 Local.var - Declare New Function Blocks.

2020-08-06
NtParam.typ - Add Two Actions (NtParamSave and NtParamLoad) - Export and import NtParam in XML Format
NtParam Act Main, Act_Initial, tyNtParam, InitLocal, Local.var and InputRef.var - Add The Additional Actions Related Variables
TLBuz - All Act_Backgrounds Change Manual Mode Towerlight To Cater For Error Indication
LFLeader - Add More Tags For Improving Leader Follower Concept, Modify p_diReqProdWidth To Use Downstream Width
LFFollower, Follower 1 	- Add fbOnlineChk For Leader Online Status
						- Modify Act_Initial,Act_Background, Act_Background_AccData
						- Add eCurrMachineStat For Status Indication
ProdRcp.typ		- Add second width
LibVer - Act_Main - Modify LibVerActReadChk, Add Step To Check File Validity.
		 Local.var - Add Alarm Text For File Coruption.

2020-07-24
MagRcp -  Add One Action in Act Main - MagRcpActSort
ProdRcp, MagRcp - p_sSearch and sSearch in Local changed to STRING[254]
ProdRcp, MagRcp - sRcpNm for RcpParam in both ProdRcp.typ and MagRcp.typ temporary changed to STRING[30]

2020-06-30
Revert Traverser Main.st and AWClose Background.st program.
Add Estun error code "65362: sAxisErrTxt := 'Torque output alarm'";

2020-06-08
ProdRcp - Increase Product Recipe Name Length to 254, Add Two Actions in Act Main - ProdRcpActSort & ProdRcpActEndCharFilter
LibVer - Act_Main - LibVerActReadChk, made error if library data files corrupted.

2020-06-05
MagConv - Update the Status of Mag Conv.Add one Action - MagConvActEntToMid.

2020-06-01
Stepper - New package for stepper control.
MotorBrk - Renewed package. Added MotorBrkActSetMtrDirOrCCW1 and MotorBrkActRstMtrDirOrCCW1.
	 	 - Modified fbRotCW and fbRotCCW and the access type to fbConvSenToSenBrkTm2Lmt.
	 	 - Added diMtrSigOnDlyTm (500), diMtrDirOffDlyTm (500), diMtrBrkOnDlyTm(100).

2020-04-28
MagConv - Add MagConvActEntToMid Action.

2020-03-20
NtParam  - Add the selection of Motor model.

2020-03-16
TLBuz - Add two inputs for buzzer behaviour, towerlight flash function to act_background and reset fbwarning.

2019-12-24
LFLeader - Remove fbBlkDS2 in Act_Initial & Act_Background_Process, add pa_bLFOnline in Act_Background_Process

2019-10-31
TLBuz - Regroup Structure Into Nutek, Aptiv & MEK.
MagConv - Separate Program Into MagConv1Clamper & MagConv2Clamper.

2019-10-21
MagConv - Improve with Action MagConvActPreExit & MagConvActPreExitClpr.
LFFollower - Improve Change All Function Without Manually Accept Data.
LFLeader - Add Second Oven Index, Improve Change All Function Without Manually Accept Data.
OpcUaMap.uad - Enable bBypassMnlAccDat Tag Name.
Startup - Act_Main_SDOWrite, Remove SDOWrite.
CANOpenServo - Change Structure Of SDOWrite And Abnormal Movement.

2019-07-30
CANOpenServo - Due To Upgrade of NtMotion.

2019-07-18
LFFollower - Act_Link, Minor debug.

2019-07-15
LCS - Act_Link, Check Recipe Name Must Not Exceed 15 Char.

2019-07-10
LCS - Add More Parameter For Live Data.

2019-07-04
LFFollower - Improve of Recipe Compare Method For p_tyInternalReqProdRcp, tyUpdtProdRcp & tyRlsBrdProdRcpNm.

2019-07-03
LFFollower - Improve Act_Background To Check Whole Product Recipe Different Instead of Name & Width Only.
Buffer - Add p_tyBufferStat & p_tyDispBuffer And Improve For Two Program Control One Memory.

2019-06-28
USHermes - Improve of Act_Background_AccData.
DSHermes - Move of Act_Background_ChgConfig.
Buffer - Improve of bParamDiff Condition.
LCSLF - Improve of LCSActRunProd.

2019-06-27
LFFollower - Improvement To Change Name & Width To Whole Product Recipe Type.

2019-06-17
Conv - Add Two Action : ConvActEntToInOff & ConvActRevImmedStart.

2019-06-12
LFFollower - Add Act_Background_ChkRlsBrd. Improvement of Act_Background_UpdtData.
LCSLF - Add Update Data in Act_Background.

2019-06-11
TLBuz - Modify ChgRcp.
LFFollower - Improvement of UpdtData.

2019-06-10
ProdRcp - Update tyCurrRcp To a_tyCurrRcp (Array).
LFFollower - Add p_bInternalUse.
USHermes - Add p_bInternalUse.
DSHermes - Add p_bInternalUse.

2019-06-07
TLBuz - Add Warning & ChgRcp.
TCP - Add Start Code & End Code Checking.
Buffer - Improve bParamDiff. Add bFIFOOld.

2019-06-04
USHermes - Improvement At Accept Date (Act_Background_AccData).

2019-06-02
TCP - New.

2019-05-30
Hermes - Debug CheckAlive. SequenceTO Start Only After Connection Establish.
Flatstream - Debug Act_Main.
USHermes - Update Act_Link to Accept New Recipe.

2019-05-29
DVFrame - Change From RS232. Improvement & Debug.
Flatstream - New.

2019-05-28
MagConv - Add MagConvActInitClpStop.
DCConv - Improvement of DC Motor Alarm Trigger Time.
LFFollower - Improve of Act_Background.
LCS - Add "Warning" & "Info" For Live Data.

2019-05-27
LFFollower - Debug Act_Link.
LCS - Debug Act_Link. Add sErrMsg.
Buffer - Debug Act_Main_Bffr. Add bMagRemoved.
Data - Update of Default User.dat.

2019-05-24
LFFollower - Improve of Act_Background.
MagConv - Add MagConvActEntClpStop.
TLBuz - Modify Warning Condition.

2019-05-22
OpcUaMap.uad - Update Tag Name.
LF - Modify Set Time. Improve Of Act_Background for Accept Data.
LFLeader - Add New Tag Name.
Time - Update of Act_InitGlobal For LF Sync Time.
LCS - Update To Reset If Receive Idle From LCS.

2019-05-21
RS232 - Add FullReadUntilValid.
LCS - Move Some Program From Act_Background To Act_Link. Bug Fixed.

2019-05-20
RS232 - Modify to work with start code & end code.
ProdRcp - Modify on dtLastModified in Act_LinkAction.
LCS - Act_Background Show Boolean & dtLastModified Working Sample. Add Function Enable.
TLBuz - Add Aptiv Mode.

2019-05-18
Buffer - Check Next Unload Ignore Product Name.

2019-05-15
OvenInfo - Improve of Act_Background.
Buffer - Add bParamDiff to check current parameter and request parameter different.

2019-05-14
LCS - Update Act_InitGlobal.
RS232 - New.

2019-05-11
LFFollower - Improve And Able To Ignore MagRcp If Necessary.

2019-05-10
TLBuz - Add Simulation Mode.
ProdRcp - Improve Act_LinkAction.
Buffer - Improve Act_LinkAction.
HWInfo - Improve Act_Main While In Simulation.

2019-05-09
CANOpenServo - Improve of Error Axis Move Abnormally By External Force (10000).
ProdRcp - Debug Write Recipe. Add Save List.
MagRcp - Debug Write Recipe. Add Save List.
UsrFolder - Create LCS Directory.
Startup - Act_Main_UsrFolder, Create LCS Directory.
Alarm - Combine Two Alarm Info.

2019-05-08
RmtHermes - Debug Log title.
UsrMgmt - Add Access Right Output.

2019-05-07
MagConv - Debug.
ConvBffr - Add Individual Have Board Output.
LF - Major update.
LCSLF - Change Name to tyCurrProdRcp.
ProdRcp - Add Write Recipe Parameter.
MagRcp - Add Write Recipe Parameter.
LCS - Update to match LCS (PC).

2019-05-04
MagRcp - Split Current Magazine Recipe From McParam.
ProdRcp - Split Current Product Recipe From McParam.
UsrMgmt - Split Access Right From McParam. Remove Nutek User.
Hermes - Split Configuration From McParam. Add RmtHermes.
Startup - Split Parameters From McParam. Add RmtHermes.
Remove "File Device" "NutekUser". Please Refer Configuration "4PPC30_043F_21F001".

2019-05-01
Hermes - Log file change to day instead of hour. Due to startup too long to check old log when production run for long.

2019-04-30
LCS - Improve To Match LCS (PC).
LFLeader - Make a_tyFollowerToLeaderTag as Output.
All - sStatTxt & a_sStatText Change To String[200].
ProdRcp - Modify For LCS.

2019-04-28
MpProdRcp - New.
Add "Config.mprecipexml" Under Configuration View > mapp. Please Refer Configuration "4PPC30_043F_21F001".
Add "File devices" For "MpProdRcp". Please Refer Configuration "4PPC30_043F_21F001".
Startup - Modify Due To MpProdRcp.

2019-04-27
DSSMEMA - Update due to NtSMEMA upgrade.

2019-04-26
Buffer - Debug tyBuffer to p_tyBuffer. Improve bLastProductUnload Condition In Unload Board.
Startup - Get Retain ConvBffr.
ConvBffr - Update Link with Startup. Improve bLastProduct Condition In Remove Board. Add Have Board Output.
LFFollower - Improve Act_LinkEn. Add Condition in Act_Link to update current recipe into leader tag.

2019-04-25
LibVer - Modify To Move LibVer From "Private" To "User".
Update "File devices" For "LibVer". Please Refer Configuration "4PPC30_043F_21F001".
Add "File devices" For "LCS". Please Refer Configuration "4PPC30_043F_21F001".
Modify "FTP Server" "Users". Please Refer Configuration "4PPC30_043F_21F001".
Modify "OpcUaMap.uad". Please Refer Configuration "4PPC30_043F_21F001".
LFLeader - Improvement.

2019-04-24
CANOpenServo - Add actual limit sensor output.
ProdRcp - Add "Add" & "Edit" action. Improve of Act_LinkAction to suit LCS.
LCS - New.

2019-04-23
LFLeader - New.

2019-04-21
USHermes - Modify Alarm Info.
LFFollower - New.

2019-04-18
ConvBffr - New.
Buffer - Change of NtBffr.

2019-04-17
CANOpenServo - Remove Extra Homing Parameter, All Use Under tyMotionCANParamInHm.

2019-04-16
Operations - Remove Accept Data & New Data.
Hermes - Debug Log File. Modify Accept Data.

2019-04-11
USHermes - Debug Log by adding step. Add p_bAccDataRdy.
DSHermes - Debug Log by adding step.

2019-04-10
Startup - bNtSettingsLoadDone should be FALSE as default.

2019-04-09
Ops2 - Update of p_bAccDat interlock by Ops1.
USHermes - Update AccDatStep in Act_Link. Remove p_bChkBrdAvl. eStatus2 = Error then bRdyRcv = false. Update Act_Background_BoardAvailableChk. Add Manual Accept Data.
DSHermes - Make local.var BoardAvailable new board parameter to default value.
NtParam - Change of Act_LinkAction.
TLBuz - Change of Act_LinkAction.
Buffer - Change of Act_LinkAction.
Conv - Change of Act_LinkAction.
DCConv - Change of Act_LinkAction.
MagConv - Change of Act_LinkAction.
MotorBrk - Change of Act_LinkAction.
ConvSpd - Change of Act_LinkAction.
SMEMA - Change of Act_LinkAction.
Pneu - Change of Act_LinkAction.
CANOpenServo - Change of Act_LinkAction.
Hermes - Change of Act_LinkAction.

2019-04-08
DSHermes - Minor debug on fbParseBrdAvlExternal.
Hermes - Add program Hermes for board available memory use.
Startup - Due to change of Hermes.

2019-04-04
OvenInfo - Add p_bBGRun.
Startup - Change eStartupStep member order for better display in UI.
UsrMgmt - Add UsrMgmtActUsrBypassLogin & UsrMgmtActNtBypassLogin.
DSHermes - Debug BoardAvailable for "New" and "External".
UI - Remove Not Use Page.

2019-03-29
All - Add Act_LinkAction.

2019-03-28
Startup - Change "DelOldLogFile" to "Alarm". Add "Hermes". Error will reset Action to IDLE.

2019-03-25
All - Change Action become input. Merge Alarm Text & Recovery Text into one type.

2019-03-22
Startup - Add bNtSettingsLoadDone. Move StartupStepParameter after StartupStepUsrFolder in Act_Main.st.
All - Update to match latest method of NtParam.

2019-03-16
Startup - Act_Main_Bffr. Add BufferActBGStartCoolFan in Step 8.

2019-03-15
Hermes - New Release

2019-03-13
UsrFolder - Debug of Log directory path. Add "FileDevice" for "Log".

2019-03-11
DCConv - Minor debug.

2019-02-26
AWClose - Minor debug.

2019-02-23
Alarm - Minor debug.
UsrFolder - Add Create Log Directory.
Startup - Improve of "Act_Main_UsrFolder" due to UsrFolder update.

2019-02-22
CANOpenServo - Change of Act_Action.

2019-02-21
DOutput - Add Act_Link.

2019-02-20
DCConv - Debug of ConvEngage.
CANOpenServo - fbModuleOK delay time change to 5s.

2019-02-19
CANOpenServo - Reset Error need to reset control word 6040.
TLBuz - Improve of condition while p_bManual = True.

2019-02-18
Buffer - Add background control of cool fan run.

2019-02-15
Conv - Improve of condition while p_bManual = True.
DCConv - Improve of condition while p_bManual = True.
MagConv - Improve of condition while p_bManual = True.
MotorBrk - Improve of condition while p_bManual = True.
SMEMA - Improve of condition while p_bManual = True.

2019-02-14
ConvSpd - Improve of condition while p_bManual = TRUE.
Change of Cyclic Time.
CANOpenServo - Change of Position Different Threshold.
Convert Library Into Binary

2019-02-11
TLBuz - Warning Rest Time Change To 5s.
Buffer - Add Magazine Present Timer.

2019-01-27
Buffer - Add error code.

2019-01-26
Buffer - Debug.

2019-01-25
Buffer - Debug a_bSkip array size.
Lifter - Debug Act_Background.
User.dat & NtUser.dat update.

2019-01-24
Pneu - Modify Cyclic for disable.
AW - Add GoWidthOff to turn off motor after auto width move.
Lifter - Debug.
Traverser - Debug.
Buffer - Debug. Add background update display.
OvenInfo - Modify Act_Main_Disable.

2019-01-23
Lifter - Major debug in slot calculation. Add FullMovRel.
CANOpenServo - Debug reset error. Debug Act_Alarm.
DCConv - Debug reset error.
Machine - Debug reset error.
Operation - Debug reset error.

2019-01-22
CANOpenServo - Minor debug.

2019-01-21
DInput - Debug reset error.
CANOpenServo - Add eMainStatus. Add bJogging.
Time - Add eMainStatus.
Operations - Rename eStatus & udiStatus.

2019-01-20
Operations - Update Structure.
SMEMA - Update due to Library update.
Buffer - Add error code.

2019-01-19
TLBuz - Add Warning.

2019-01-18
RstErr - Act_Main update.
CANOpenServo - Add output. Set Default Value for siModOfOptDisp_6061:=6.
Change of Cyclic time.
Buffer - Update Local.var
Add file for NtUser, LibrariesVersion & User.
Conv - Add Pneu status output.
DCConv - Add Pneu status output.
Operations - Modify structure in Cyclic.

2019-01-17
DCConv - Act_Main debug.

2019-01-16
Trav - Remove diPitch.
Lifter - Remove diPitch.
Operations - Modify Reset methos.

2019-01-15
McParam - File name as input.
NtParam - File name as input.
Buffer - File name as input.
Operations - Add bAccData.

2019-01-14
Operations - Update Alarm & Sequence.
SMEMA - bTimer & bVirtual as output. Debug Act_Background timer interlock.

2019-01-12
Conv - Convert time out type.
DCConv - Convert time out type.
MagConv - Convert time out type.
OvenInfo - diBrdInOven change to retain.
SMEMA - Update timer condition. Add bComplSigOn.
Startup - Debug for HWInfo.

2019-01-11
SMEMA - Minor debug. Add Act_LinkEn.
Operations - Add alarm. Add Act_LinkEn.
MagRcp - Add Act_LinkEn.
OvenInfo - Add Act_LinkEn. Minor debug.
Conv - Add Act_LinkEn. Add conveyor time out.
DCConv - Add Act_LinkEn. Add conveyor time out.
MagConv - Add Act_LinkEn. Add conveyor time out.
MotorBrk - Add Act_LinkEn.
ConvSpd - Add Act_LinkEn.
RS232Mirtec - Add Act_LinkEn.
Pneu - Add Act_LinkEn.
CANOpenServo - Add Act_LinkEn. Major Update.

2019-01-10
McParam - Remove ProdRcpWrite & MagRcpWrite.
OvenInfo - Act_Main modify for change of eStat.
Conv - Act_Main modify for change of eStat.
DCConv - Act_Main modify for change of eStat.
MagConv - Act_Main modify for change of eStat.
MotorBrk - Act_Main modify for change of eStat.
ConvSpd - Act_Main modify for change of eStat.
SMEMA - Act_Main modify for change of eStat.
DOutput - Act_Main modify for change of eStat.
Pneu - Act_Main modify for change of eStat.
Operations - Act_Main modify for change of eStat.

2019-01-09
AW - Update bWidthPosDiff when disable.
Lifter - Update bSltPosDiff when disable.
Conv - Add bGdBrdInit. Debug tMtrOffDlyTm. Improve Act_Action to let eStatus = DONE also able change eStat directly.
DCConv - Add bGdBrdInit. Improve Act_Action to let eStatus = DONE also able change eStat directly.
SMEMA - Add tRstDlyTm. Improve Act_Action to let eStatus = DONE also able change eStat directly.
Operations - Add Act_Main_Disable. Improve Act_Action to let eStatus = DONE also able change eStat directly.
TLBuz - Improve Act_Action to let eStatus = DONE also able change eStat directly.
OvenInfo - Improve Act_Action to let eStatus = DONE also able change eStat directly.
MagConv - Improve Act_Action to let eStatus = DONE also able change eStat directly.
MotorBrk - Improve Act_Action to let eStatus = DONE also able change eStat directly.
ConvSpd - Improve Act_Action to let eStatus = DONE also able change eStat directly.
DOutput - Improve Act_Action to let eStatus = DONE also able change eStat directly.
Pneu - Improve Act_Action to let eStatus = DONE also able change eStat directly.

2019-01-08 //Until Here////
DOutput - Add output.
SMEMA - bTimer will be trigger only during SMEMAActRun.
Operations - Combine Ops1 & Ops2 into Ops.

2019-01-07
SMEMA - Add bUSRdy, bUSGdBrdRdy & bDSRdy for USSMEMA & DSSMEMA.
Conv - Add tMtrOffDlyTm.
DCConv - Add tMtrOffDlyTm.
MagConv - Add tMtrOffDlyTm.
Time - Combine Error
CANOpenServo - Combine Error
Alarm - Remove link data.

2019-01-04
Machine - Debug Act_Alarm1.
Time - Debug Init.st.
Operations - Debug Ops1 > Act_Main. Add sStepTxt into Act_Main. Add Act_Dummy.
Conv - Due to NtConv update, add one more type of Exit.
DCConv - Due to NtConv update, add one more type of Exit.
MagConv - Due to NtConv update, add one more type of Exit.
SMEMA - Add Timer & Virtual.

2019-01-03
Machine - Debug Act_Alarm & Act_Alarm1. Modify background error handling.
CANOpenServo - Modify background error handling. Update sStatTxt in Act_Initial.
AW - Replace diStandPitchInUM (Input) to diPitchInUM (Local).
Time - Modify background error handling. Update sStatTxt in Act_Initial.
DCConv - Modify background error handling. Update sStatTxt in Act_Initial.
DInput - Modify background error handling.
UsrMgmt - Update sStatTxt in Act_Initial.
McParam - Update sStatTxt in Act_Initial.
NtParam - Update sStatTxt in Act_Initial.
ProdRcp - Update sStatTxt in Act_Initial.
MagRcp - Update sStatTxt in Act_Initial.
HWInfo - Update sStatTxt in Act_Initial.
UsrFolder - Update sStatTxt in Act_Initial.
LibVer - Update sStatTxt in Act_Initial.
General - Update sStatTxt in Act_Initial.
TLBuz - Update sStatTxt in Act_Initial.
OvenInfo - Update sStatTxt in Act_Initial.
Buffer - Update sStatTxt in Act_Initial.
RstErr - Update sStatTxt in Act_Initial.
Conv - Update sStatTxt in Act_Initial.
MagConv - Update sStatTxt in Act_Initial.
MotorBrk - Update sStatTxt in Act_Initial.
ConvSpd - Update sStatTxt in Act_Initial.
Alarm - Update sStatTxt in Act_Initial.
RS232Mirtec - Update sStatTxt in Act_Initial.
SMEMA - Update sStatTxt in Act_Initial.
UI - Update sStatTxt in Act_Initial.
DOutput - Update sStatTxt in Act_Initial.
Pneu - Update sStatTxt in Act_Initial.
Operations - Update sStatTxt in Act_Initial.
Startup - Update sStatTxt in Act_Initial.

2019-01-02
UsrMgmt - Change of sStatTxt update.
McParam - Change of sStatTxt update.
NtParam - Change of sStatTxt update.
ProdRcp - Change of sStatTxt update.
MagRcp - Change of sStatTxt update.
Time - Change of sStatTxt update.
HWInfo - Change of sStatTxt update.
UsrFolder - Change of sStatTxt update.
LibVer - Change of sStatTxt update.
General - Change of sStatTxt update.
TLBuz - Change of sStatTxt update.
OvenInfo - Change of sStatTxt update.
Buffer - Change of sStatTxt update.
RstErr - Change of sStatTxt update.
Conv - Change of sStatTxt update.
DCConv - Change of sStatTxt update.
MagConv - Change of sStatTxt update.
MotorBrk - Change of sStatTxt update.
ConvSpd - Change of sStatTxt update.
Alarm - Change of sStatTxt update.
RS232Mirtec - Change of sStatTxt update.
SMEMA - Change of sStatTxt update.
UI - Change of sStatTxt update.
DOutput - Change of sStatTxt update.
Pneu - Change of sStatTxt update.
Operations - Change of sStatTxt update.
CANOpenServo - Change of sStatTxt update. Update eStatus to Busy while running.
Startup - Change of sStatTxt update.

2018-12-31
CANOpenServo - Seperate input reference.

2018-12-27
Time - Remove bBGRun.
TLBuz - Remove bBGRun. Add manual reset.
OvenInfo - Background direct link to input bPrepExtdd, bEnExtdd & bDisExtdd. Add manual reset.
Buffer - Background Cool Fan Control direct link to input bPrepCoolTm & bCoolFanTm.
DCConv - Remove bBGRun. Add manual reset.
AlarmLog - Background run is control by Action.
Machine - Remove bBGRun.
SMEMA - Remove bBGRun. Add manual reset.
DInput - Remove bBGRun.
DOutput - Remove bBGRun. Add manual reset.
CANOpenServo - Remove bBGRun. Background run is control by Action. Add manual reset.
AW - Add bWidthPosDiff.
Lifter - Add bSltPosDiff.
Startup - Background run is control by Action. Shorten local variable name.
McParam - Add McParam program without Magazine (McParam2).
RstErr - Add manual reset.
Conv - Add manual reset.
MagConv - Add manual reset.
MotorBrk - Add manual reset.
ConvSpd - Add manual reset.
Pneu - Add manual reset.

2018-12-26
CPU - Update distribute of program in CPU. Update cyclic time.
FTP - Update of FTP server configurations.
Startup - Remove bStartupErr.
HWInfo - After set new IPAddr & Subnetmask will update output.
TLBuz - Rising of bManual will set Amber Light ON.
Conv - Remove functions reset in individual eStat.
MagConv - Remove functions reset in individual eStat.
MotorBrk - Remove functions reset in individual eStat.
DCConv - New program.
Operations - Update of OperationsActStep.

2018-12-24
Operations - Add bRun.Sequence will execute base on bRun instead of bStatusRun.

2018-12-21
Buffer - Add individual cooling fan control.
McParam - Move Hermes parameter to Hermes program type.
MagConv - Add bClprTwoOutputControl. Remove bClprUnclampCtrl.

2018-12-20
TLBuz - Add bMuteBuz.
OvenInfo - Add bDis.
Conv - Add bEn.
MagConv - Add bEn.
MotorBrk - Add bEn.
ConvSpd - Add bEn.
RS232Mirtec - Add bEn.
SMEMA - Add bDis.
Pneu - Add bEn.
CANOpenServo - Add bEn.
CANOpenServo - AutoWidth - Add diMaxWidthInUM, diMinWidthInUM, diWidthOffsetInUM & diStdPitch.
Operations - Add bPrep, bEn & bDis. Add OperationsStatusCycleStopping. Default Status is OperationsStatusStop. Add Boolean output for Status.
MagRcp - Change sDisplayInfo & Magazine Parameter.
Startup - Add bRun.

2018-12-14
RstErr - Add bManual to control reset of output in Idle. Reset output in Idle after ManualMode off.
Conv - Add bManual to control reset of output in Idle. Rename eAction. Reset output in Idle after ManualMode off.
ConvSpd - Add bManual to control reset of output in Idle. Reset output in Idle after ManualMode off.
MtrBrk - Add bManual to control reset of output in Idle. Rename eAction. Reset output in Idle after ManualMode off. Reset after change eStat.
MagConv - Add bManual to control reset of output in Idle. Rename eAction. Reset output in Idle after ManualMode off. Reset after change eStat.
OvenInfo - Set bOvenAllow to TRUE, if all functions not activated.
SMEMA - Reset output in Idle after ManualMode off.
Pneu - Add Extended & Retracted output.

2018-12-13
Conv - Change of Conv2Sen to Conv. Add Reject & Inspection functions. Add individual output control.
Pneu - Add bTwoCtrlIn & bTwoCtrlOut.
TLBuz - Add individual output control.
ConvSpd - Add individual output control.
OvenInfo - Add individual output control. Move functions into Act_Background.
RstErr - Add individual output control.
MtrBrk - Add individual output control.
MagConv - Add individual output control.
DOutput - Add individual output control.
SMEMA - Add individual output control.

2018-12-12
Startup - Add Logout during User Management Startup.
Time - Move Act_Background above Act_Main.
Buffer - Move Act_Background above Act_Main.
Alarm - Move Act_Background above Act_Main.
CANOpenServo - Move Act_Background above Act_Main.
Operations - Change of Conv2Sen to Conv.

2018-12-11
DOutput - Split to Act_InitGlobal & Act_InitLocal.
Pneu - Change in all program. Add Pneu3Sen program.
Operations - Update sample to 2 operations. Rename variable.
CANOpenServo - Rename variable.
```

- LibrariesVersion.dat (binary file, 2222 bytes)
### SoftwareVersion.var
```iecst
VAR CONSTANT
	sSWVersion : STRING[30] := 'NAEUL004C00R14L518F00';
END_VAR
```

### Library Logical/NtLibraries/NtGeneral (IEC, version 5.00.1) - 5.00.1 - Add tyAlmTxt
5.00.0 - New Library Design. (20181211)

#### Types.typ - Exported data types
```iecst
(*Library Status*)

TYPE
	eFBStatus :
		( (*Function Block Status*)
		Idle, (*Library In Idle Status*)
		Done, (*Library In Done Status*)
		Busy, (*Library In Busy Status*)
		Error (*Library In Error Status*)
		);
END_TYPE

(**)
(*Alarm*)

TYPE
	tyAlmTxt : 	STRUCT
		sAlmText : STRING[200]; (*Alarm Text*)
		sRcyText : STRING[200]; (*Recovery Text*)
	END_STRUCT;
	tyAlmDat : 	STRUCT
		udiCode : UDINT; (*Alarm Code*)
		eSeverity : eAlmSeverity; (*Alarm Severity*)
		udiRunTime : UDINT; (*Run Time*)
		udiModuleNum : UDINT;
		bAlm : BOOL;
		bWarning : BOOL;
	END_STRUCT;
	eAlmSeverity :
		(
		AlmSeverityNA, (*Error*)
		AlmSeverityError, (*Error*)
		AlmSeverityWarning, (*Warning*)
		AlmSeverityInfo (*Information*)
		);
	tyAlmInputProps : 	STRUCT
		uiModuleOrder : UINT;
	END_STRUCT;
END_TYPE

(*Others*)

TYPE
	tyValidCharChkrInternal : {REDUND_UNREPLICABLE} 	STRUCT  (*Local Variables*)
		sValidChar : {REDUND_UNREPLICABLE} STRING[1]; (*Valid Characters For Checking*)
		sCharChk : {REDUND_UNREPLICABLE} STRING[1]; (*Character On Checking*)
		i : {REDUND_UNREPLICABLE} INT;
		j : {REDUND_UNREPLICABLE} INT;
	END_STRUCT;
	tyInvalidCharChkrInternal : {REDUND_UNREPLICABLE} 	STRUCT  (*Local Variables*)
		sInvalidChar : {REDUND_UNREPLICABLE} STRING[1]; (*Invalid Characters For Checking*)
		sCharChk : {REDUND_UNREPLICABLE} STRING[1]; (*Character On Checking*)
		i : {REDUND_UNREPLICABLE} INT;
		j : {REDUND_UNREPLICABLE} INT;
	END_STRUCT;
	tyCheckDuplicateInternal : {REDUND_UNREPLICABLE} 	STRUCT  (*Local Variables*)
		i : {REDUND_UNREPLICABLE} USINT;
		j : {REDUND_UNREPLICABLE} USINT;
		usiCnt : {REDUND_UNREPLICABLE} USINT; (*Counter*)
	END_STRUCT;
	tyStringSearchInternal : {REDUND_UNREPLICABLE} 	STRUCT  (*Local Variables*)
		i : {REDUND_UNREPLICABLE} UDINT;
		usiZero : {REDUND_UNREPLICABLE} USINT; (*Counter*)
	END_STRUCT;
	tyCheckExistInternal : {REDUND_UNREPLICABLE} 	STRUCT  (*Local Variables*)
		i : {REDUND_UNREPLICABLE} USINT;
		j : {REDUND_UNREPLICABLE} USINT;
		usiCnt : {REDUND_UNREPLICABLE} USINT; (*Counter*)
	END_STRUCT;
	tySenFltrInternal : {REDUND_UNREPLICABLE} 	STRUCT  (*Local Variables*)
		fbSigFltrTm : {REDUND_UNREPLICABLE} TON; (*Signal Filter Time*)
	END_STRUCT;
	tyIPValidInternal : 	STRUCT  (*Local Variables*)
		i : INT;
		iCnt : INT; (*Counter*)
		a_iDotPos : ARRAY[1..3]OF INT; (*IP Address Dot Position*)
		a_sIPPart : ARRAY[1..4]OF STRING[3]; (*IP Address Part in String*)
		a_iIPPart : ARRAY[1..4]OF INT; (*IP Address Part in Integer*)
		sMismatchChar : STRING[1]; (*Mismatch Character*)
	END_STRUCT;
END_TYPE
```

### Library Logical/NtLibraries/NtUI (IEC, version 5.00.2) - 5.00.2 - Add tyUIBitmap & tyUIBtn (uiValueIdx) to accomodate higher range of offset index (20210625)
5.00.1 - Update fbTableCtrl, fbTableCtrl_v2 and tyUILString.(20200608)
5.00.0 - New Library Design. (20181203)

#### Types.typ - Exported data types
```iecst
TYPE
	tyTouchGetActionInternal : 	STRUCT  (*Local Variables*)
		udiHandle : UDINT; (*Visu Handle*)
		tyTouchAction : TouchAction; (*Output of Touch Action*)
	END_STRUCT;
	tyTouchFilterInternal : 	STRUCT  (*Local Variables*)
		udiXOld : UDINT; (*Old Coordinate X Value*)
		udiYOld : UDINT; (*Old Coordinate Y Value*)
	END_STRUCT;
	tyTouchGetSlideDistInternal : 	STRUCT  (*Local Variables*)
		fbPressedRise : R_TRIG; (*Rising Edge of Press Action*)
		fbInternalPressedRise : R_TRIG; (*Internal Rising Edge of Press Action*)
		bValidStartPress : BOOL; (*Valid of Start Press*)
		bPressed : BOOL; (*Touchscreen Pressed*)
		udiXTemp : UDINT; (*Temporary Coordinate X*)
		udiYTemp : UDINT; (*Temporary Coordinate Y*)
	END_STRUCT;
	tyTouchGetTapInternal : 	STRUCT  (*Local Variables*)
		fbInternalPressedRise : R_TRIG; (*Internal Rising Edge of Press Action*)
		fbInternalPressedFall : F_TRIG; (*Internal Falling Edge of Press Action*)
		bPressed : BOOL; (*Touchscreen Pressed*)
		tTmTemp : TIME; (*Time of Temporary*)
		udiXTemp : UDINT; (*Temporary Coordinate X*)
		udiYTemp : UDINT; (*Temporary Coordinate Y*)
		tTmPrev : TIME; (*Time of Previous*)
		udiXPrev : UDINT; (*Previous Coordinate X*)
		udiYPrev : UDINT; (*Previous Coordinate Y*)
	END_STRUCT;
	tyTableCtrlInternal : 	STRUCT  (*Local Variables*)
		fbSingleTapChkDlyTm : TON; (*Single Tap Check Delay Time*)
		fbSliderOffTm : TON; (*Slider Off Time*)
		fbSelectedRowMnlRise : R_TRIG; (*Rising Edge of Manual Select Row*)
		fbTablePosUpRise : R_TRIG; (*Rising Edge of Up Table Position*)
		fbTablePosDownRise : R_TRIG; (*Rising Edge of Down Table Position*)
		fbSliderRelease : F_TRIG; (*Falling Edge of Slider Active*)
		fbTouchFilter : fbTouchFilter;
		fbTouchGetAction : fbTouchGetAction;
		fbTouchGetSlideDist : fbTouchGetSlideDist;
		fbTouchGetTap : fbTouchGetTap;
		i : INT;
		iTablePos : INT; (*Table Position*)
		iTablePosTemp : INT; (*Temporary Table Position*)
	END_STRUCT;
END_TYPE

(**)
(*Basic Controls*)

TYPE
	tyUILine : 	STRUCT  (*UI Line*)
		uiMaskRtStat : UINT := 1; (*Mask Status Datapoint*)
		uiRtStat : UINT := 0; (*Status Datapoint*)
		usiColor : USINT := 0; (*Color Datapoint*)
	END_STRUCT;
	tyUITxt : 	STRUCT  (*UI Text*)
		bHighlighting : BOOL := FALSE; (*Highlighting Datapoint*)
		sTxt : STRING[30] := ''; (*Text Datapoint*)
		uiMaskRtStat : UINT := 1; (*Mask Status Datapoint*)
		uiRtStat : UINT := 0; (*Status Datapoint*)
		usiColor : USINT := 0; (*Color Datapoint*)
		usiValueIdx : USINT := 0; (*Value Index Datapoint*)
	END_STRUCT;
	tyUIAlmTxt : 	STRUCT  (*UI Text*)
		bHighlighting : BOOL := FALSE; (*Highlighting Datapoint*)
		sTxt : STRING[30] := ''; (*Text Datapoint*)
		uiMaskRtStat : UINT := 1; (*Mask Status Datapoint*)
		uiRtStat : UINT := 0; (*Status Datapoint*)
		usiColor : USINT := 0; (*Color Datapoint*)
		udiValueIdx : UDINT := 0; (*Value Index Datapoint*)
	END_STRUCT;
	tyUIShape : 	STRUCT  (*UI Shape*)
		uiMaskRtStat : UINT := 1; (*Mask Status Datapoint*)
		uiRtStat : UINT := 0; (*Status Datapoint*)
		usiColor : USINT := 0; (*Color Datapoint*)
	END_STRUCT;
	tyUIString : 	STRUCT  (*UI String*)
		bRtCompl : BOOL := FALSE; (*Completion Datapoint*)
		bRtLk : BOOL := FALSE; (*Locking Datapoint*)
		sValue : STRING[30] := ''; (*Value Datapoint*)
		sValueDisplay : STRING[10] := ''; (*Value Datapoint*)
		uiMaskRtStat : UINT := 1; (*Mask Status Datapoint*)
		uiRtStat : UINT := 0; (*Status Datapoint*)
		usiColor : USINT := 0; (*Color Datapoint*)
		sKeypadTitle : STRING[30]; (*Keypad Title*)
	END_STRUCT;
	tyUILString : 	STRUCT  (*UI String*)
		bRtCompl : BOOL := FALSE; (*Completion Datapoint*)
		bRtLk : BOOL := FALSE; (*Locking Datapoint*)
		sValue : STRING[254] := ''; (*Value Datapoint*)
		uiMaskRtStat : UINT := 1; (*Mask Status Datapoint*)
		uiRtStat : UINT := 0; (*Status Datapoint*)
		usiColor : USINT := 0; (*Color Datapoint*)
		sKeypadTitle : STRING[30]; (*Keypad Title*)
		udiValueIdx : UDINT;
	END_STRUCT;
	tyUINum : 	STRUCT  (*UI Numeric*)
		bRtCompl : BOOL := FALSE; (*Completion Datapoint*)
		bRtLk : BOOL := FALSE; (*Locking Datapoint*)
		diValue : DINT := 0; (*Value Datapoint*)
		diValueMax : DINT := 0; (*Max Value Datapoint*)
		diValueMin : DINT := 0; (*Min Value Datapoint*)
		diValueTeach : DINT := 0; (*Teach Value Datapoint*)
		uiMaskRtStat : UINT := 1; (*Mask Status Datapoint*)
		uiRtStat : UINT := 0; (*Status Datapoint*)
		usiAddDigits : USINT := 0; (*Add Fraction Digits Datapoint*)
		usiColor : USINT := 0; (*Color Datapoint*)
		sKeypadTitle : STRING[30]; (*Keypad Title*)
	END_STRUCT;
	tyUIBtn : 	STRUCT  (*UI Button*)
		bRtCompl : BOOL := FALSE; (*Completion Datapoint*)
		bRtLk : BOOL := FALSE; (*Locking Datapoint*)
		bValue : BOOL := FALSE; (*Boolean Value Datapoint*)
		uiMaskRtStat : UINT := 1; (*Mask Status Datapoint*)
		uiRtStat : UINT := 0; (*Status Datapoint*)
		usiBitmapIdx : USINT := 0; (*Bitmap Index Datapoint*)
		usiColor : USINT := 0; (*Color Datapoint*)
		usiPressedColor : USINT := 0; (*Button Pressed Color Datapoint*)
		usiTxtIdx : USINT := 0; (*Text Index Datapoint*)
		uiBitmapIdx : UINT := 0; (*Bitmap Index Datapoint*)
	END_STRUCT;
	tyUIHotspot : 	STRUCT  (*UI Hotspot*)
		bRtCompl : BOOL := FALSE; (*Completion Datapoint*)
		bRtLk : BOOL := FALSE; (*Locking Datapoint*)
		bValue : BOOL := FALSE; (*Boolean Value Datapoint*)
		uiMaskRtStat : UINT := 1; (*Mask Status Datapoint*)
		uiRtStat : UINT := 0; (*Status Datapoint*)
	END_STRUCT;
	tyUIBitmap : 	STRUCT  (*UI Bitmap*)
		uiMaskRtStat : UINT := 1; (*Mask Status Datapoint*)
		uiRtStat : UINT := 0; (*Status Datapoint*)
		usiColor : USINT := 0; (*Color Datapoint*)
		usiValueIdx : USINT := 0; (*Value Index Datapoint*)
		uiValueIdx : UINT := 0; (*Value Index Datapoint*)
	END_STRUCT;
	tyUIBarGraph : 	STRUCT  (*UI Bar Graph*)
		iValue : INT := 0; (*Value Datapoint*)
		uiMaskRtStat : UINT := 1; (*Mask Status Datapoint*)
		uiRtStat : UINT := 0; (*Status Datapoint*)
		usiColor : USINT := 0; (*Color Datapoint*)
	END_STRUCT;
	tyUIDT : 	STRUCT  (*UI DateTime*)
		diValue : DINT := 0; (*Value Datapoint*)
		uiMaskRtStat : UINT := 1; (*Mask Status Datapoint*)
		uiRtStat : UINT := 0; (*Status Datapoint*)
		usiColor : USINT := 0; (*Color Datapoint*)
	END_STRUCT;
	tyUIPw : 	STRUCT  (*UI Password*)
		a_sTxt : ARRAY[0..9]OF STRING[30] := [10('')]; (*Text Datapoint*)
		bRtCompl : BOOL := FALSE; (*Completion Datapoint*)
		bRtLk : BOOL := FALSE; (*Locking Datapoint*)
		uiMaskRtStat : UINT := 1; (*Mask Status Datapoint*)
		uiRtStat : UINT := 0; (*Status Datapoint*)
		usiColor : USINT := 0; (*Color Datapoint*)
		usiLevel : USINT := 0; (*Level Datapoint*)
	END_STRUCT;
	tyUIListBox : 	STRUCT  (*UI List Box*)
		a_sTxt : ARRAY[0..9]OF STRING[30] := [10('')]; (*Text Datapoint*)
		a_usiValueOptionIdx : ARRAY[0..9]OF USINT := [10(0)]; (*Option Value Index Datapoint*)
		bRtCompl : BOOL := FALSE; (*Completion Datapoint*)
		bRtLk : BOOL := FALSE; (*Locking Datapoint*)
		uiMaskRtStat : UINT := 1; (*Mask Status Datapoint*)
		uiRtStat : UINT := 0; (*Status Datapoint*)
		usiColor : USINT := 0; (*Color Datapoint*)
		usiDisabledColor : USINT := 0; (*Disabled Color Datapoint*)
		usiSelectedColor : USINT := 0; (*Selected Color Datapoint*)
		usiSliderColor : USINT := 0; (*Slider Color Datapoint*)
		usiValueIdx : USINT := 0; (*Value Index Datapoint*)
		usiValueMaxIdx : USINT := 0; (*Max Value Index Datapoint*)
		usiValueMinIdx : USINT := 0; (*Min Value Index Datapoint*)
	END_STRUCT;
	tyUIAlm : 	STRUCT  (*UI Alarm*)
		a_usiFltrTm : ARRAY[0..5]OF USINT := [6(0)]; (*Filter Time Datapoint*)
		bRtLk : BOOL := FALSE; (*Locking Datapoint*)
		uiMaskRtStat : UINT := 1; (*Mask Status Datapoint*)
		uiRtStat : UINT := 0; (*Status Datapoint*)
		usiColor : USINT := 0; (*Color Datapoint*)
		uiFltrAlm : UINT := 0; (*Filter Alarm Datapoint*)
		uiFltrCtrl : UINT := 0; (*Filter Control Datapoint*)
		uiFltrGrp : UINT := 0; (*Filter Group Datapoint*)
		uiFltrPriority : UINT := 0; (*Filter Priority Datapoint*)
	END_STRUCT;
	tyUIDrawBox : 	STRUCT  (*UI Draw Box*)
		uiMaskRtStat : UINT := 1; (*Mask Status Datapoint*)
		uiRtStat : UINT := 0; (*Status Datapoint*)
	END_STRUCT;
	tyUITrend : 	STRUCT  (*UI Trend*)
		bRtCompl : BOOL := FALSE; (*Completion Datapoint*)
		bRtLk : BOOL := FALSE; (*Locking Datapoint*)
		iSelectItem : INT := 0; (*Select Item Datapoint*)
		uiMaskRtStat : UINT := 1; (*Mask Status Datapoint*)
		uiRtStat : UINT := 0; (*Status Datapoint*)
		usiColor : USINT := 0; (*Color Datapoint*)
	END_STRUCT;
	tyUIScale : 	STRUCT  (*UI Scale*)
		iMaxValue : INT := 0; (*Max Value Datapoint*)
		iMinValue : INT := 0; (*Min Value Datapoint*)
		iRangeEnd : INT := 0; (*Range End Datapoint*)
		iRangeSt : INT := 0; (*Range Start Datapoint*)
		iValue : INT := 0; (*Value Datapoint*)
		uiMaskRtStat : UINT := 1; (*Mask Status Datapoint*)
		uiRtStat : UINT := 0; (*Status Datapoint*)
		usiColor : USINT := 0; (*Color Datapoint*)
		usiRangeColor : USINT := 0; (*Range Color Datapoint*)
	END_STRUCT;
	tyUIEdit : 	STRUCT  (*UI Edit*)
		bLineEndings : BOOL := FALSE; (*Line Endings Datapoint*)
		bRtCompl : BOOL := FALSE; (*Completion Datapoint*)
		bRtEditInsertMode : BOOL := FALSE; (*Edit Insert Mode Datapoint*)
		bRtEditModified : BOOL := FALSE; (*Edit Modified Datapoint*)
		bRtEditSelectionMode : BOOL := FALSE; (*Edit Selection Mode Datapoint*)
		bRtLk : BOOL := FALSE; (*Locking Datapoint*)
		iRtEditCursorColumn : INT := 0; (*Edit Cursor Column Datapoint*)
		iRtEditCursorLine : INT := 0; (*Edit Cursor Line Datapoint*)
		sRtCmdRequest : STRING[30] := ''; (*Command Request Datapoint*)
		sRtCmdResponse : STRING[30] := ''; (*Command Response Datapoint*)
		sURL : STRING[30] := ''; (*URL Datapoint*)
		sValue : STRING[30] := ''; (*Value Datapoint*)
		uiMaskRtStat : UINT := 1; (*Mask Status Datapoint*)
		uiRtBusy : UINT := 0; (*Busy Datapoint*)
		uiRtCmdStat : UINT := 0; (*Command Status Datapoint*)
		uiRtStat : UINT := 0; (*Status Datapoint*)
		usiColor : USINT := 0; (*Color Datapoint*)
		usiCursorColor : USINT := 0; (*Cursor Color Datapoint*)
		usiSelectedColor : USINT := 0; (*Selected Color Datapoint*)
	END_STRUCT;
	tyUIHTMLView : 	STRUCT  (*UI HTML View*)
		bRtLk : BOOL := FALSE; (*Locking Datapoint*)
		sChgURL : STRING[30] := ''; (*Change URL Datapoint*)
		sCurrTitle : STRING[30] := ''; (*Current Title Datapoint*)
		sCurrURL : STRING[30] := ''; (*Current URL Datapoint*)
		sHTMLStream : STRING[30] := ''; (*HTML Stream*)
		uiMaskRtStat : UINT := 1; (*Mask Status Datapoint*)
		uiRtBusy : UINT := 0; (*Busy Datapoint*)
		uiRtHTTPErrCode : UINT := 0; (*HTTP Error Code*)
		uiRtStat : UINT := 0; (*Status Datapoint*)
		usiColor : USINT := 0; (*Color Datapoint*)
		usiErrCnt : USINT := 0; (*Error Count Datapoint*)
	END_STRUCT;
	tyUIDrpDn : 	STRUCT  (*UI Dropdown*)
		a_usiValueOptionIdx : ARRAY[0..9]OF USINT := [10(0)]; (*Option Value Index Datapoint*)
		bRtCompl : BOOL := FALSE; (*Completion Datapoint*)
		bRtLk : BOOL := FALSE; (*Locking Datapoint*)
		sTxt : STRING[30] := ''; (*Text Datapoint*)
		uiMaskRtStat : UINT := 1; (*Mask Status Datapoint*)
		uiRtStat : UINT := 0; (*Status Datapoint*)
		usiColor : USINT := 0; (*Color Datapoint*)
		usiDisabledColor : USINT := 0; (*Disabled Color Datapoint*)
		usiDropdownColor : USINT := 0; (*Dropdown Color Datapoint*)
		usiSelectedColor : USINT := 0; (*Selected Color Datapoint*)
		usiValueIdx : USINT := 0; (*Value Index Datapoint*)
		usiValueMaxIdx : USINT := 0; (*Max Value Index Datapoint*)
		usiValueMinIdx : USINT := 0; (*Min Value Index Datapoint*)
	END_STRUCT;
	tyUIPieChart : 	STRUCT  (*UI Pie Chart*)
		a_uiValue : ARRAY[0..9]OF UINT := [10(0)]; (*Value Datapoint*)
		uiMaskRtStat : UINT := 1; (*Mask Status Datapoint*)
		uiRtStat : UINT := 0; (*Status Datapoint*)
		usiColor : USINT := 0; (*Color Datapoint*)
	END_STRUCT;
	tyUISlider : 	STRUCT  (*UI Slider*)
		bRtCompl : BOOL := FALSE; (*Completion Datapoint*)
		bRtLk : BOOL := FALSE; (*Locking Datapoint*)
		iCurrValue : INT := 0; (*Current Value Datapoint*)
		iMaxValue : INT := 0; (*Max Value Datapoint*)
		iMinValue : INT := 0; (*Min Value Datapoint*)
		iValue : INT := 0; (*Value Datapoint*)
		uiMaskRtStat : UINT := 1; (*Mask Status Datapoint*)
		uiRtStat : UINT := 0; (*Status Datapoint*)
		usiColor : USINT := 0; (*Color Datapoint*)
	END_STRUCT;
	tyUIGauge : 	STRUCT  (*UI Gauge*)
		iMaxValue : INT := 0; (*Max Value Datapoint*)
		iMinValue : INT := 0; (*Min Value Datapoint*)
		iValue : INT := 0; (*Value Datapoint*)
		uiMaskRtStat : UINT := 1; (*Mask Status Datapoint*)
		uiRtStat : UINT := 0; (*Status Datapoint*)
		usiColor : USINT := 0; (*Color Datapoint*)
	END_STRUCT;
	tyUITable : 	STRUCT  (*UI Table*)
		a_tyHotspot : ARRAY[1..15]OF tyUIHotspot; (*Array Of Hotspot*)
		a_tyStringDataCol0 : ARRAY[1..15]OF tyUILString; (*Array Of Number Listing (column: 0 / x = 0)*)
		a_tyStringDataCol1 : ARRAY[1..15]OF tyUILString; (*Array Of Data (column: 1 / x = 1)*)
		a_tyStringDataCol2 : ARRAY[1..15]OF tyUILString; (*Array Of Data (column: 2 / x = 2)*)
		a_tyStringDataCol3 : ARRAY[1..15]OF tyUILString; (*Array Of Data (column: 3 / x = 3)*)
		a_tyStringDataCol4 : ARRAY[1..15]OF tyUILString; (*Array Of Data (column: 4 / x = 4)*)
		tyUISlider : tyUISlider := (uiRtStat:=1); (*Scroll Bar Scale*)
		tyStringTitle0Col0Row0 : tyUIString; (*Number Listing Title (row: 0, column: 0 / x = 0, y = 0)*)
		tyStringTitle1Col1Row0 : tyUIString; (*Title (row: 0, column: 1 / x = 1, y = 0)*)
		tyStringTitle2Col2Row0 : tyUIString; (*Title (row: 0, column: 2 / x = 2, y = 0)*)
		tyStringTitle3Col3Row0 : tyUIString; (*Title (row: 0, column: 3 / x = 3, y = 0)*)
		tyStringTitle4Col4Row0 : tyUIString; (*Title (row: 0, column: 4 / x = 4, y = 0)*)
		uiMaskRtStat : UINT := 1; (*Mask Status Datapoint*)
	END_STRUCT;
	tyUITable1 : 	STRUCT  (*UI Table*)
		a_tyHotspot : ARRAY[1..15]OF tyUIHotspot; (*Array Of Hotspot*)
		a_tyStringDataCol0 : ARRAY[1..15]OF tyUILString; (*Array Of Number Listing (column: 0 / x = 0)*)
		a_tyStringDataCol1 : ARRAY[1..15]OF tyUILString; (*Array Of Data (column: 1 / x = 1)*)
		a_tyStringDataCol2 : ARRAY[1..15]OF tyUILString; (*Array Of Data (column: 2 / x = 2)*)
		a_tyStringDataCol4 : ARRAY[1..15]OF tyUILString; (*Array Of Data (column: 4 / x = 4)*)
		a_tyTxtDataCol3 : ARRAY[1..15]OF tyUITxt; (*Array Of Data (column: 3 / x = 3)*)
		tyStringTitle0Col0Row0 : tyUIString; (*Number Listing Title (row: 0, column: 0 / x = 0, y = 0)*)
		tyStringTitle1Col1Row0 : tyUIString; (*Title (row: 0, column: 1 / x = 1, y = 0)*)
		tyStringTitle2Col2Row0 : tyUIString; (*Title (row: 0, column: 2 / x = 2, y = 0)*)
		tyStringTitle3Col3Row0 : tyUIString; (*Title (row: 0, column: 3 / x = 3, y = 0)*)
		tyStringTitle4Col4Row0 : tyUIString; (*Title (row: 0, column: 4 / x = 4, y = 0)*)
		tyUISlider : tyUISlider := (uiRtStat:=1); (*Scroll Bar Scale*)
		uiMaskRtStat : UINT := 1; (*Mask Status Datapoint*)
	END_STRUCT;
	tyUILyr : 	STRUCT  (*UI Layer*)
		uiRtStat : UINT := 0; (*Status Datapoint*)
	END_STRUCT;
	tyUIAlarm : 	STRUCT
		tyUIAlmCur : tyAlm;
		tyUIAlmHis : tyAlm;
	END_STRUCT;
	tyAlm : 	STRUCT
		usiColor : USINT;
		udiCntrllDp : INT;
		udiGrpDp : UDINT;
		udiAlrmDp : UDINT;
		udiPrioDp : UDINT;
		udiTimeDp : DATE_AND_TIME;
		uiRtStat : UINT;
	END_STRUCT;
	tyUIAlarmInfoGrp : 	STRUCT
		udiOffsetInfo1 : UDINT;
		udiOffsetInfo2 : UDINT;
		tyUptTxtSnipp : tyUIAlmTextSnip;
		udiToggleAlarmInfo : UDINT;
	END_STRUCT;
	tyUIAlmTextSnip : 	STRUCT
		CurrentRecipeName : STRING[80];
		CurrentRecipeWidth : STRING[80];
		SameRcpDiffWidName : STRING[80];
		MachineOutGoingWidth : STRING[80];
		LFNewRecipeName : STRING[80];
		LFNewRecipeWidth : STRING[80];
		LFOldRecipeName : STRING[80];
		LFOldRecipeWidth : STRING[80];
		HANewRecipeName : STRING[80];
		HANewRecipeWidth : STRING[80];
		HAOldRecipeName : STRING[80];
		HAOldRecipeWidth : STRING[80];
		HBNewRecipeName : STRING[80];
		HBNewRecipeWidth : STRING[80];
		HBOldRecipeName : STRING[80];
		HBOldRecipeWidth : STRING[80];
	END_STRUCT;
END_TYPE
```

### Library Logical/NtLibraries/NtOpConXML (IEC, version 5.00.0) - 5.00.1 - Added plcGrab with 3 magazine presence. (20230707)
5.00.0 - New LIbrary Design (20230510)

#### Types.typ - Exported data types
```iecst
(*Message Type*)

TYPE
	tyOpConMsgType : 	STRUCT
		bEventRcv : BOOL;
		bPlcGrabRcv : BOOL;
		bPartRcvRetCode : BOOL; (*Check Alive*)
		bTypeNo : BOOL; (*Check Alive Ping*)
		bTypeVar : BOOL; (*Check Alive Pong*)
		reserve1 : BOOL; (*Service Description*)
		reserve2 : BOOL; (*Notification*)
	END_STRUCT;
	eOpConMsgType :
		(
		OpConMsgTypeNA, (*NA*)
		OpConMsgTypeEventReceived,
		OpConMsgTypePartReceived,
		OpConMsgTypePlcGrabReceived,
		OpConMsgTypePartProcessed,
		OpConMsgTypePLCError,
		OpConMsgTypePartMissingStarted,
		OpConMsgTypePartMissing,
		OpConMsgTypePLCJamStarted,
		OpConMsgTypePLCJam,
		OpConMsgTypePLCGrab
		);
END_TYPE

(**)
(*opCon Full Data*)

TYPE
	tyEventType : 	STRUCT
		tyData : tyEventTypeData;
		tyAvl : tyEventTypeAvl;
	END_STRUCT;
	tyLocationParam : 	STRUCT
		tyData : tyLocationParamData;
		tyAvl : tyLocationParamAvl;
	END_STRUCT;
	tyOpConPartReceive : 	STRUCT
		tyData : tyPartReceiveData;
		tyAvl : tyPartReceiveAvl;
	END_STRUCT;
	tyOpConPlcGrabReceive : 	STRUCT
		tyData : tyPlcGrabReceiveData;
		tyAvl : tyPlcGrabReceiveAvl;
	END_STRUCT;
	tyOpConPartProcessed : 	STRUCT
		tyData : tyPartProcessedData;
		tyAvl : tyPartProcessedAvl;
	END_STRUCT;
	tyOpConPLCError : 	STRUCT
		tyData : tyPLCErrorData;
		tyAvl : tyPLCErrorAvl;
	END_STRUCT;
	tyOpConPartMissing : 	STRUCT
		tyData : tyPartMissingData;
		tyAvl : tyPartMissingAvl;
	END_STRUCT;
	tyOpConPLCJam : 	STRUCT
		tyData : tyPLCJamData;
		tyAvl : tyPLCJamAvl;
	END_STRUCT;
	tyOpConPLCGrab : 	STRUCT
		tyData : tyPLCGrabData;
		tyAvl : tyPLCGrabAvl;
	END_STRUCT;
END_TYPE

(**)
(*opCon Message Data*)

TYPE
	tyEventTypeData : 	STRUCT
		uiEventId : UINT;
		sVersion : STRING[5];
		sEventName : STRING[30];
		siEventSwitch : SINT;
		usiContentType : USINT;
	END_STRUCT;
	tyLocationParamData : 	STRUCT
		uiLineNo : UINT;
		uiStatNo : UINT;
		uiStatIdx : UINT;
		uiFuNo : UINT;
		uiWorkPos : UINT;
		uiToolPos : UINT;
		sProcessName : STRING[30];
		uiProcessNo : UINT;
		sApplication : STRING[5];
	END_STRUCT;
	tyPlcGrabReceiveData : 	STRUCT
		iReturnCode : INT;
		sTraceTxt : STRING[254];
		sLevel : STRING[20];
		reserve1 : USINT;
		reserve2 : USINT;
		reserve3 : USINT;
	END_STRUCT;
	tyPartReceiveData : 	STRUCT
		sIdentifier : STRING[254];
		sTypeNo : STRING[20];
		sTypeVar : STRING[4];
		asName : STRING[30];
		asDataType : STRING[2];
		asValue : STRING[254];
		iReturnCode : INT;
		sTraceTxt : STRING[254];
		reserve2 : USINT;
	END_STRUCT;
	tyPartProcessedData : 	STRUCT
		sIdentifier : STRING[254];
		usiResult : USINT;
		sTypeNo : STRING[20];
		sTypeVar : STRING[4];
		usiWorkingCode : USINT;
		usiNioBits : USINT;
		uiBatch : USINT;
		sMachineID : STRING[5];
		sName : ARRAY[0..4]OF STRING[30];
		sDataType : ARRAY[0..4]OF STRING[2];
		sValue : ARRAY[0..4]OF STRING[254];
	END_STRUCT;
	tyPLCErrorData : 	STRUCT
		sTypeNo : STRING[20];
		sTypeVar : STRING[4];
		uiErrorNo : UINT;
		sErrorText : STRING[254];
		usiErrorType : USINT;
		usiErrorState : USINT;
		usiOperationMode : USINT;
		bModeOn : BOOL;
		iChainNo : INT;
	END_STRUCT;
	tyPartMissingData : 	STRUCT
		usiMissingPart : USINT;
		sTypeNo : STRING[20];
		sTypeVar : STRING[4];
	END_STRUCT;
	tyPLCJamData : 	STRUCT
		sTypeNo : STRING[20];
		sTypeVar : STRING[4];
	END_STRUCT;
	tyPLCGrabData : 	STRUCT
		sMagazineNm : ARRAY[0..4]OF STRING[30];
		sValue : ARRAY[0..4]OF STRING[10];
		sDataType : ARRAY[0..4]OF STRING[2];
	END_STRUCT;
END_TYPE

(**)
(*opCon Data Availability*)

TYPE
	tyEventTypeAvl : 	STRUCT
		bEventId : BOOL;
		bVersion : BOOL;
		bEventName : BOOL;
		bEventSwitch : BOOL;
		bContentType : BOOL;
		bIdentifier : BOOL;
		bTypeNo : BOOL;
		bTypeVar : BOOL;
		bName : BOOL;
		bValue : BOOL;
		reserve1 : BOOL;
		reserve2 : BOOL;
		reserve3 : BOOL;
		reserve4 : BOOL;
	END_STRUCT;
	tyLocationParamAvl : 	STRUCT
		bLineNo : BOOL;
		bStatNo : BOOL;
		bStatIdx : BOOL;
		bFuNo : BOOL;
		bWorkPos : BOOL;
		bToolPos : BOOL;
		bProcessName : BOOL;
		bProcessNo : BOOL;
		bApplication : BOOL;
	END_STRUCT;
	tyPlcGrabReceiveAvl : 	STRUCT
		bIdentifier : BOOL;
		bTypeNo : BOOL;
		bTypeVar : BOOL;
		bName : BOOL;
		bDataType : BOOL;
		bValue : BOOL;
		bReturnCode : BOOL;
		bTraceTxt : BOOL;
		reserve2 : BOOL;
	END_STRUCT;
	tyPartReceiveAvl : 	STRUCT
		bIdentifier : BOOL;
		bTypeNo : BOOL;
		bTypeVar : BOOL;
		bName : BOOL;
		bDataType : BOOL;
		bValue : BOOL;
		bReturnCode : BOOL;
		bTraceTxt : BOOL;
		reserve2 : BOOL;
	END_STRUCT;
	tyPartProcessedAvl : 	STRUCT
		bIdentifier : BOOL;
		bResult : BOOL;
		bTypeNo : BOOL;
		bTypeVar : BOOL;
		bWorkingCode : BOOL;
		bNioBits : BOOL;
		bBatch : BOOL;
		bMachineID : BOOL;
		bName : ARRAY[0..4]OF BOOL;
		bDataType : ARRAY[0..4]OF BOOL;
		bValue : ARRAY[0..4]OF BOOL;
	END_STRUCT;
	tyPLCErrorAvl : 	STRUCT
		bTypeNo : BOOL;
		bTypeVar : BOOL;
		bErrorNo : BOOL;
		bErrorText : BOOL;
		bErrorType : BOOL;
		bErrorState : BOOL;
		bOperationMode : BOOL;
		bModeOn : BOOL;
		bChainNo : BOOL;
	END_STRUCT;
	tyPartMissingAvl : 	STRUCT
		bMissingPart : BOOL;
		bTypeNo : BOOL;
		bTypeVar : BOOL;
	END_STRUCT;
	tyPLCJamAvl : 	STRUCT
		bTypeNo : BOOL;
		bTypeVar : BOOL;
	END_STRUCT;
	tyPLCGrabAvl : 	STRUCT
		bMagazineNm : ARRAY[0..4]OF BOOL;
		bValue : ARRAY[0..4]OF BOOL;
		bDataType : ARRAY[0..4]OF BOOL;
	END_STRUCT;
END_TYPE
```
